LIN {X -176.622,Y -112.343,Z 160.000,A 0.000,B 0.000,C 180.000,E1 0.000} C_DIS
LIN {X -182.169,Y -103.103,Z 160.000,A 0.000,B 0.000,C 180.000,E1 0.000} C_DIS
LIN {X -187.236,Y -93.587,Z 160.000,A 0.000,B 0.000,C 180.000,E1 0.000} C_DIS
LIN {X -191.804,Y -83.827,Z 160.000,A 0.000,B 0.000,C 180.000,E1 0.000} C_DIS
LIN {X -195.867,Y -73.837,Z 160.000,A 0.000,B 0.000,C 180.000,E1 0.000} C_DIS
LIN {X -199.408,Y -63.658,Z 160.000,A 0.000,B 0.000,C 180.000,E1 0.000} C_DIS
LIN {X -202.421,Y -53.309,Z 160.000,A 0.000,B 0.000,C 180.000,E1 0.000} C_DIS
LIN {X -204.896,Y -42.818,Z 160.000,A 0.000,B 0.000,C 180.000,E1 0.000} C_DIS
LIN {X -206.829,Y -32.213,Z 160.000,A 0.000,B 0.000,C 180.000,E1 0.000} C_DIS
LIN {X -208.213,Y -21.523,Z 160.000,A 0.000,B 0.000,C 180.000,E1 0.000} C_DIS
LIN {X -208.336,Y -19.932,Z 160.000,A 0.000,B 0.000,C 180.000,E1 0.000} C_DIS
LIN {X 19.906,Y 208.310,Z 160.000,A 0.000,B 0.000,C 180.000,E1 0.000} C_DIS
;rapid-leaky
$VEL.CP=0.3
LIN {X -233.236,Y -36.326,Z 170.000,A 0.000,B 0.000,C 180.000,E1 0.000} C_DIS
;bead-perimeter_outer
$VEL.CP=0.59
LIN {X -231.057,Y -48.285,Z 170.000,A 0.000,B 0.000,C 180.000,E1 0.000} C_DIS
LIN {X -228.265,Y -60.113,Z 170.000,A 0.000,B 0.000,C 180.000,E1 0.000} C_DIS
LIN {X -224.866,Y -71.785,Z 170.000,A 0.000,B 0.000,C 180.000,E1 0.000} C_DIS
LIN {X -220.874,Y -83.267,Z 170.000,A 0.000,B 0.000,C 180.000,E1 0.000} C_DIS
LIN {X -216.295,Y -94.525,Z 170.000,A 0.000,B 0.000,C 180.000,E1 0.000} C_DIS
LIN {X -211.142,Y -105.535,Z 170.000,A 0.000,B 0.000,C 180.000,E1 0.000} C_DIS
LIN {X -205.429,Y -116.265,Z 170.000,A 0.000,B 0.000,C 180.000,E1 0.000} C_DIS
LIN {X -199.171,Y -126.685,Z 170.000,A 0.000,B 0.000,C 180.000,E1 0.000} C_DIS
LIN {X -192.385,Y -136.770,Z 170.000,A 0.000,B 0.000,C 180.000,E1 0.000} C_DIS
LIN {X -185.089,Y -146.493,Z 170.000,A 0.000,B 0.000,C 180.000,E1 0.000} C_DIS
LIN {X -177.303,Y -155.828,Z 170.000,A 0.000,B 0.000,C 180.000,E1 0.000} C_DIS
LIN {X -169.045,Y -164.748,Z 170.000,A 0.000,B 0.000,C 180.000,E1 0.000} C_DIS
LIN {X -160.340,Y -173.232,Z 170.000,A 0.000,B 0.000,C 180.000,E1 0.000} C_DIS
LIN {X -151.211,Y -181.256,Z 170.000,A 0.000,B 0.000,C 180.000,E1 0.000} C_DIS
LIN {X -141.679,Y -188.800,Z 170.000,A 0.000,B 0.000,C 180.000,E1 0.000} C_DIS
LIN {X -131.772,Y -195.844,Z 170.000,A 0.000,B 0.000,C 180.000,E1 0.000} C_DIS
LIN {X -121.516,Y -202.367,Z 170.000,A 0.000,B 0.000,C 180.000,E1 0.000} C_DIS
LIN {X -110.937,Y -208.354,Z 170.000,A 0.000,B 0.000,C 180.000,E1 0.000} C_DIS
LIN {X -100.064,Y -213.788,Z 170.000,A 0.000,B 0.000,C 180.000,E1 0.000} C_DIS
LIN {X -88.925,Y -218.657,Z 170.000,A 0.000,B 0.000,C 180.000,E1 0.000} C_DIS
LIN {X -77.552,Y -222.945,Z 170.000,A 0.000,B 0.000,C 180.000,E1 0.000} C_DIS
LIN {X -65.972,Y -226.641,Z 170.000,A 0.000,B 0.000,C 180.000,E1 0.000} C_DIS
LIN {X -54.217,Y -229.736,Z 170.000,A 0.000,B 0.000,C 180.000,E1 0.000} C_DIS
LIN {X -42.318,Y -232.223,Z 170.000,A 0.000,B 0.000,C 180.000,E1 0.000} C_DIS
LIN {X -30.307,Y -234.093,Z 170.000,A 0.000,B 0.000,C 180.000,E1 0.000} C_DIS
LIN {X -18.217,Y -235.343,Z 170.000,A 0.000,B 0.000,C 180.000,E1 0.000} C_DIS
LIN {X -6.078,Y -235.969,Z 170.000,A 0.000,B 0.000,C 180.000,E1 0.000} C_DIS
LIN {X 6.078,Y -235.969,Z 170.000,A 0.000,B 0.000,C 180.000,E1 0.000} C_DIS
LIN {X 17.057,Y -235.404,Z 170.000,A 0.000,B 0.000,C 180.000,E1 0.000} C_DIS
LIN {X 18.215,Y -235.344,Z 170.000,A 0.000,B 0.000,C 180.000,E1 0.000} C_DIS
LIN {X 30.307,Y -234.093,Z 170.000,A 0.000,B 0.000,C 180.000,E1 0.000} C_DIS
LIN {X 42.318,Y -232.223,Z 170.000,A 0.000,B 0.000,C 180.000,E1 0.000} C_DIS
LIN {X 54.217,Y -229.736,Z 170.000,A 0.000,B 0.000,C 180.000,E1 0.000} C_DIS
LIN {X 65.972,Y -226.641,Z 170.000,A 0.000,B 0.000,C 180.000,E1 0.000} C_DIS
LIN {X 77.552,Y -222.945,Z 170.000,A 0.000,B 0.000,C 180.000,E1 0.000} C_DIS
LIN {X 88.925,Y -218.657,Z 170.000,A 0.000,B 0.000,C 180.000,E1 0.000} C_DIS
LIN {X 100.064,Y -213.788,Z 170.000,A 0.000,B 0.000,C 180.000,E1 0.000} C_DIS
LIN {X 110.937,Y -208.354,Z 170.000,A 0.000,B 0.000,C 180.000,E1 0.000} C_DIS
LIN {X 121.516,Y -202.367,Z 170.000,A 0.000,B 0.000,C 180.000,E1 0.000} C_DIS
LIN {X 131.772,Y -195.844,Z 170.000,A 0.000,B 0.000,C 180.000,E1 0.000} C_DIS
LIN {X 141.679,Y -188.800,Z 170.000,A 0.000,B 0.000,C 180.000,E1 0.000} C_DIS
LIN {X 151.211,Y -181.256,Z 170.000,A 0.000,B 0.000,C 180.000,E1 0.000} C_DIS
LIN {X 160.340,Y -173.232,Z 170.000,A 0.000,B 0.000,C 180.000,E1 0.000} C_DIS
LIN {X 169.045,Y -164.748,Z 170.000,A 0.000,B 0.000,C 180.000,E1 0.000} C_DIS
LIN {X 177.303,Y -155.828,Z 170.000,A 0.000,B 0.000,C 180.000,E1 0.000} C_DIS
LIN {X 185.089,Y -146.493,Z 170.000,A 0.000,B 0.000,C 180.000,E1 0.000} C_DIS
LIN {X 192.385,Y -136.770,Z 170.000,A 0.000,B 0.000,C 180.000,E1 0.000} C_DIS
LIN {X 199.171,Y -126.685,Z 170.000,A 0.000,B 0.000,C 180.000,E1 0.000} C_DIS
LIN {X 205.429,Y -116.265,Z 170.000,A 0.000,B 0.000,C 180.000,E1 0.000} C_DIS
LIN {X 211.142,Y -105.535,Z 170.000,A 0.000,B 0.000,C 180.000,E1 0.000} C_DIS
LIN {X 216.295,Y -94.525,Z 170.000,A 0.000,B 0.000,C 180.000,E1 0.000} C_DIS
LIN {X 220.874,Y -83.267,Z 170.000,A 0.000,B 0.000,C 180.000,E1 0.000} C_DIS
LIN {X 224.866,Y -71.785,Z 170.000,A 0.000,B 0.000,C 180.000,E1 0.000} C_DIS
LIN {X 228.265,Y -60.113,Z 170.000,A 0.000,B 0.000,C 180.000,E1 0.000} C_DIS
LIN {X 231.057,Y -48.285,Z 170.000,A 0.000,B 0.000,C 180.000,E1 0.000} C_DIS
LIN {X 233.236,Y -36.326,Z 170.000,A 0.000,B 0.000,C 180.000,E1 0.000} C_DIS
LIN {X 234.796,Y -24.271,Z 170.000,A 0.000,B 0.000,C 180.000,E1 0.000} C_DIS
LIN {X 235.735,Y -12.151,Z 170.000,A 0.000,B 0.000,C 180.000,E1 0.000} C_DIS
LIN {X 236.047,Y 0.000,Z 170.000,A 0.000,B 0.000,C 180.000,E1 0.000} C_DIS
LIN {X 235.735,Y 12.151,Z 170.000,A 0.000,B 0.000,C 180.000,E1 0.000} C_DIS
LIN {X 234.796,Y 24.271,Z 170.000,A 0.000,B 0.000,C 180.000,E1 0.000} C_DIS
LIN {X 233.236,Y 36.326,Z 170.000,A 0.000,B 0.000,C 180.000,E1 0.000} C_DIS
LIN {X 231.057,Y 48.285,Z 170.000,A 0.000,B 0.000,C 180.000,E1 0.000} C_DIS
LIN {X 228.265,Y 60.113,Z 170.000,A 0.000,B 0.000,C 180.000,E1 0.000} C_DIS
LIN {X 224.866,Y 71.785,Z 170.000,A 0.000,B 0.000,C 180.000,E1 0.000} C_DIS
LIN {X 220.874,Y 83.267,Z 170.000,A 0.000,B 0.000,C 180.000,E1 0.000} C_DIS
LIN {X 216.295,Y 94.525,Z 170.000,A 0.000,B 0.000,C 180.000,E1 0.000} C_DIS
LIN {X 211.142,Y 105.535,Z 170.000,A 0.000,B 0.000,C 180.000,E1 0.000} C_DIS
LIN {X 205.429,Y 116.265,Z 170.000,A 0.000,B 0.000,C 180.000,E1 0.000} C_DIS
LIN {X 199.171,Y 126.685,Z 170.000,A 0.000,B 0.000,C 180.000,E1 0.000} C_DIS
LIN {X 192.385,Y 136.770,Z 170.000,A 0.000,B 0.000,C 180.000,E1 0.000} C_DIS
LIN {X 185.089,Y 146.493,Z 170.000,A 0.000,B 0.000,C 180.000,E1 0.000} C_DIS
LIN {X 177.303,Y 155.828,Z 170.000,A 0.000,B 0.000,C 180.000,E1 0.000} C_DIS
LIN {X 169.045,Y 164.748,Z 170.000,A 0.000,B 0.000,C 180.000,E1 0.000} C_DIS
LIN {X 160.340,Y 173.232,Z 170.000,A 0.000,B 0.000,C 180.000,E1 0.000} C_DIS
LIN {X 151.211,Y 181.256,Z 170.000,A 0.000,B 0.000,C 180.000,E1 0.000} C_DIS
LIN {X 141.679,Y 188.800,Z 170.000,A 0.000,B 0.000,C 180.000,E1 0.000} C_DIS
LIN {X 131.772,Y 195.844,Z 170.000,A 0.000,B 0.000,C 180.000,E1 0.000} C_DIS
LIN {X 121.516,Y 202.367,Z 170.000,A 0.000,B 0.000,C 180.000,E1 0.000} C_DIS
LIN {X 110.937,Y 208.354,Z 170.000,A 0.000,B 0.000,C 180.000,E1 0.000} C_DIS
LIN {X 100.064,Y 213.788,Z 170.000,A 0.000,B 0.000,C 180.000,E1 0.000} C_DIS
LIN {X 88.925,Y 218.657,Z 170.000,A 0.000,B 0.000,C 180.000,E1 0.000} C_DIS
LIN {X 77.552,Y 222.945,Z 170.000,A 0.000,B 0.000,C 180.000,E1 0.000} C_DIS
LIN {X 65.972,Y 226.641,Z 170.000,A 0.000,B 0.000,C 180.000,E1 0.000} C_DIS
LIN {X 54.217,Y 229.736,Z 170.000,A 0.000,B 0.000,C 180.000,E1 0.000} C_DIS
LIN {X 42.318,Y 232.223,Z 170.000,A 0.000,B 0.000,C 180.000,E1 0.000} C_DIS
LIN {X 30.307,Y 234.093,Z 170.000,A 0.000,B 0.000,C 180.000,E1 0.000} C_DIS
LIN {X 18.217,Y 235.343,Z 170.000,A 0.000,B 0.000,C 180.000,E1 0.000} C_DIS
LIN {X 6.078,Y 235.969,Z 170.000,A 0.000,B 0.000,C 180.000,E1 0.000} C_DIS
LIN {X -6.078,Y 235.969,Z 170.000,A 0.000,B 0.000,C 180.000,E1 0.000} C_DIS
LIN {X -18.215,Y 235.344,Z 170.000,A 0.000,B 0.000,C 180.000,E1 0.000} C_DIS
LIN {X -30.307,Y 234.093,Z 170.000,A 0.000,B 0.000,C 180.000,E1 0.000} C_DIS
LIN {X -42.318,Y 232.223,Z 170.000,A 0.000,B 0.000,C 180.000,E1 0.000} C_DIS
LIN {X -54.217,Y 229.736,Z 170.000,A 0.000,B 0.000,C 180.000,E1 0.000} C_DIS
LIN {X -65.972,Y 226.641,Z 170.000,A 0.000,B 0.000,C 180.000,E1 0.000} C_DIS
LIN {X -77.552,Y 222.945,Z 170.000,A 0.000,B 0.000,C 180.000,E1 0.000} C_DIS
LIN {X -88.925,Y 218.657,Z 170.000,A 0.000,B 0.000,C 180.000,E1 0.000} C_DIS
LIN {X -100.064,Y 213.788,Z 170.000,A 0.000,B 0.000,C 180.000,E1 0.000} C_DIS
LIN {X -110.937,Y 208.354,Z 170.000,A 0.000,B 0.000,C 180.000,E1 0.000} C_DIS
LIN {X -121.516,Y 202.367,Z 170.000,A 0.000,B 0.000,C 180.000,E1 0.000} C_DIS
LIN {X -131.772,Y 195.844,Z 170.000,A 0.000,B 0.000,C 180.000,E1 0.000} C_DIS
LIN {X -141.679,Y 188.800,Z 170.000,A 0.000,B 0.000,C 180.000,E1 0.000} C_DIS
LIN {X -151.211,Y 181.256,Z 170.000,A 0.000,B 0.000,C 180.000,E1 0.000} C_DIS
LIN {X -160.340,Y 173.232,Z 170.000,A 0.000,B 0.000,C 180.000,E1 0.000} C_DIS
LIN {X -169.045,Y 164.748,Z 170.000,A 0.000,B 0.000,C 180.000,E1 0.000} C_DIS
LIN {X -177.303,Y 155.828,Z 170.000,A 0.000,B 0.000,C 180.000,E1 0.000} C_DIS
LIN {X -185.089,Y 146.493,Z 170.000,A 0.000,B 0.000,C 180.000,E1 0.000} C_DIS
LIN {X -192.385,Y 136.770,Z 170.000,A 0.000,B 0.000,C 180.000,E1 0.000} C_DIS
LIN {X -199.171,Y 126.685,Z 170.000,A 0.000,B 0.000,C 180.000,E1 0.000} C_DIS
LIN {X -205.429,Y 116.265,Z 170.000,A 0.000,B 0.000,C 180.000,E1 0.000} C_DIS
LIN {X -211.142,Y 105.535,Z 170.000,A 0.000,B 0.000,C 180.000,E1 0.000} C_DIS
LIN {X -216.295,Y 94.525,Z 170.000,A 0.000,B 0.000,C 180.000,E1 0.000} C_DIS
LIN {X -220.874,Y 83.267,Z 170.000,A 0.000,B 0.000,C 180.000,E1 0.000} C_DIS
LIN {X -224.866,Y 71.785,Z 170.000,A 0.000,B 0.000,C 180.000,E1 0.000} C_DIS
LIN {X -228.265,Y 60.113,Z 170.000,A 0.000,B 0.000,C 180.000,E1 0.000} C_DIS
LIN {X -231.057,Y 48.285,Z 170.000,A 0.000,B 0.000,C 180.000,E1 0.000} C_DIS
LIN {X -233.236,Y 36.326,Z 170.000,A 0.000,B 0.000,C 180.000,E1 0.000} C_DIS
LIN {X -234.796,Y 24.271,Z 170.000,A 0.000,B 0.000,C 180.000,E1 0.000} C_DIS
LIN {X -235.735,Y 12.151,Z 170.000,A 0.000,B 0.000,C 180.000,E1 0.000} C_DIS
LIN {X -236.047,Y 0.000,Z 170.000,A 0.000,B 0.000,C 180.000,E1 0.000} C_DIS
LIN {X -235.735,Y -12.151,Z 170.000,A 0.000,B 0.000,C 180.000,E1 0.000} C_DIS
LIN {X -234.796,Y -24.271,Z 170.000,A 0.000,B 0.000,C 180.000,E1 0.000} C_DIS
LIN {X -233.236,Y -36.326,Z 170.000,A 0.000,B 0.000,C 180.000,E1 0.000} C_DIS
;rapid-leaky
$VEL.CP=0.3
LIN {X -217.875,Y -33.934,Z 170.000,A 0.000,B 0.000,C 180.000,E1 0.000} C_DIS
;bead-perimeter_inner
$VEL.CP=0.59
LIN {X -215.841,Y -45.105,Z 170.000,A 0.000,B 0.000,C 180.000,E1 0.000} C_DIS
LIN {X -213.232,Y -56.153,Z 170.000,A 0.000,B 0.000,C 180.000,E1 0.000} C_DIS
LIN {X -210.057,Y -67.058,Z 170.000,A 0.000,B 0.000,C 180.000,E1 0.000} C_DIS
LIN {X -206.328,Y -77.784,Z 170.000,A 0.000,B 0.000,C 180.000,E1 0.000} C_DIS
LIN {X -202.050,Y -88.300,Z 170.000,A 0.000,B 0.000,C 180.000,E1 0.000} C_DIS
LIN {X -197.237,Y -98.585,Z 170.000,A 0.000,B 0.000,C 180.000,E1 0.000} C_DIS
LIN {X -191.900,Y -108.608,Z 170.000,A 0.000,B 0.000,C 180.000,E1 0.000} C_DIS
LIN {X -186.055,Y -118.342,Z 170.000,A 0.000,B 0.000,C 180.000,E1 0.000} C_DIS
LIN {X -179.716,Y -127.763,Z 170.000,A 0.000,B 0.000,C 180.000,E1 0.000} C_DIS
LIN {X -172.900,Y -136.846,Z 170.000,A 0.000,B 0.000,C 180.000,E1 0.000} C_DIS
LIN {X -165.626,Y -145.566,Z 170.000,A 0.000,B 0.000,C 180.000,E1 0.000} C_DIS
LIN {X -157.913,Y -153.898,Z 170.000,A 0.000,B 0.000,C 180.000,E1 0.000} C_DIS
LIN {X -149.781,Y -161.824,Z 170.000,A 0.000,B 0.000,C 180.000,E1 0.000} C_DIS
LIN {X -141.253,Y -169.319,Z 170.000,A 0.000,B 0.000,C 180.000,E1 0.000} C_DIS
LIN {X -132.349,Y -176.367,Z 170.000,A 0.000,B 0.000,C 180.000,E1 0.000} C_DIS
LIN {X -123.095,Y -182.946,Z 170.000,A 0.000,B 0.000,C 180.000,E1 0.000} C_DIS
LIN {X -113.514,Y -189.039,Z 170.000,A 0.000,B 0.000,C 180.000,E1 0.000} C_DIS
LIN {X -103.631,Y -194.633,Z 170.000,A 0.000,B 0.000,C 180.000,E1 0.000} C_DIS
LIN {X -93.474,Y -199.709,Z 170.000,A 0.000,B 0.000,C 180.000,E1 0.000} C_DIS
LIN {X -83.068,Y -204.257,Z 170.000,A 0.000,B 0.000,C 180.000,E1 0.000} C_DIS
LIN {X -72.445,Y -208.262,Z 170.000,A 0.000,B 0.000,C 180.000,E1 0.000} C_DIS
LIN {X -61.628,Y -211.715,Z 170.000,A 0.000,B 0.000,C 180.000,E1 0.000} C_DIS
LIN {X -50.647,Y -214.607,Z 170.000,A 0.000,B 0.000,C 180.000,E1 0.000} C_DIS
LIN {X -39.532,Y -216.930,Z 170.000,A 0.000,B 0.000,C 180.000,E1 0.000} C_DIS
LIN {X -28.312,Y -218.677,Z 170.000,A 0.000,B 0.000,C 180.000,E1 0.000} C_DIS
LIN {X -17.017,Y -219.845,Z 170.000,A 0.000,B 0.000,C 180.000,E1 0.000} C_DIS
LIN {X -5.678,Y -220.429,Z 170.000,A 0.000,B 0.000,C 180.000,E1 0.000} C_DIS
LIN {X 5.679,Y -220.429,Z 170.000,A 0.000,B 0.000,C 180.000,E1 0.000} C_DIS
LIN {X 16.253,Y -219.885,Z 170.000,A 0.000,B 0.000,C 180.000,E1 0.000} C_DIS
LIN {X 17.011,Y -219.845,Z 170.000,A 0.000,B 0.000,C 180.000,E1 0.000} C_DIS
LIN {X 28.312,Y -218.677,Z 170.000,A 0.000,B 0.000,C 180.000,E1 0.000} C_DIS
LIN {X 39.532,Y -216.930,Z 170.000,A 0.000,B 0.000,C 180.000,E1 0.000} C_DIS
LIN {X 50.647,Y -214.607,Z 170.000,A 0.000,B 0.000,C 180.000,E1 0.000} C_DIS
LIN {X 61.628,Y -211.715,Z 170.000,A 0.000,B 0.000,C 180.000,E1 0.000} C_DIS
LIN {X 72.445,Y -208.262,Z 170.000,A 0.000,B 0.000,C 180.000,E1 0.000} C_DIS
LIN {X 83.068,Y -204.257,Z 170.000,A 0.000,B 0.000,C 180.000,E1 0.000} C_DIS
LIN {X 93.474,Y -199.709,Z 170.000,A 0.000,B 0.000,C 180.000,E1 0.000} C_DIS
LIN {X 103.631,Y -194.633,Z 170.000,A 0.000,B 0.000,C 180.000,E1 0.000} C_DIS
LIN {X 113.514,Y -189.039,Z 170.000,A 0.000,B 0.000,C 180.000,E1 0.000} C_DIS
LIN {X 123.095,Y -182.946,Z 170.000,A 0.000,B 0.000,C 180.000,E1 0.000} C_DIS
LIN {X 132.349,Y -176.367,Z 170.000,A 0.000,B 0.000,C 180.000,E1 0.000} C_DIS
LIN {X 141.253,Y -169.319,Z 170.000,A 0.000,B 0.000,C 180.000,E1 0.000} C_DIS
LIN {X 149.781,Y -161.824,Z 170.000,A 0.000,B 0.000,C 180.000,E1 0.000} C_DIS
LIN {X 157.913,Y -153.898,Z 170.000,A 0.000,B 0.000,C 180.000,E1 0.000} C_DIS
LIN {X 165.626,Y -145.566,Z 170.000,A 0.000,B 0.000,C 180.000,E1 0.000} C_DIS
LIN {X 172.900,Y -136.846,Z 170.000,A 0.000,B 0.000,C 180.000,E1 0.000} C_DIS
LIN {X 179.716,Y -127.763,Z 170.000,A 0.000,B 0.000,C 180.000,E1 0.000} C_DIS
LIN {X 186.055,Y -118.342,Z 170.000,A 0.000,B 0.000,C 180.000,E1 0.000} C_DIS
LIN {X 191.900,Y -108.608,Z 170.000,A 0.000,B 0.000,C 180.000,E1 0.000} C_DIS
LIN {X 197.237,Y -98.585,Z 170.000,A 0.000,B 0.000,C 180.000,E1 0.000} C_DIS
LIN {X 202.050,Y -88.300,Z 170.000,A 0.000,B 0.000,C 180.000,E1 0.000} C_DIS
LIN {X 206.328,Y -77.784,Z 170.000,A 0.000,B 0.000,C 180.000,E1 0.000} C_DIS
LIN {X 210.057,Y -67.058,Z 170.000,A 0.000,B 0.000,C 180.000,E1 0.000} C_DIS
LIN {X 213.232,Y -56.153,Z 170.000,A 0.000,B 0.000,C 180.000,E1 0.000} C_DIS
LIN {X 215.841,Y -45.105,Z 170.000,A 0.000,B 0.000,C 180.000,E1 0.000} C_DIS
LIN {X 217.875,Y -33.934,Z 170.000,A 0.000,B 0.000,C 180.000,E1 0.000} C_DIS
LIN {X 219.334,Y -22.672,Z 170.000,A 0.000,B 0.000,C 180.000,E1 0.000} C_DIS
LIN {X 220.210,Y -11.351,Z 170.000,A 0.000,B 0.000,C 180.000,E1 0.000} C_DIS
LIN {X 220.502,Y 0.000,Z 170.000,A 0.000,B 0.000,C 180.000,E1 0.000} C_DIS
LIN {X 220.210,Y 11.351,Z 170.000,A 0.000,B 0.000,C 180.000,E1 0.000} C_DIS
LIN {X 219.334,Y 22.672,Z 170.000,A 0.000,B 0.000,C 180.000,E1 0.000} C_DIS
LIN {X 217.875,Y 33.934,Z 170.000,A 0.000,B 0.000,C 180.000,E1 0.000} C_DIS
LIN {X 215.841,Y 45.105,Z 170.000,A 0.000,B 0.000,C 180.000,E1 0.000} C_DIS
LIN {X 213.232,Y 56.153,Z 170.000,A 0.000,B 0.000,C 180.000,E1 0.000} C_DIS
LIN {X 210.057,Y 67.058,Z 170.000,A 0.000,B 0.000,C 180.000,E1 0.000} C_DIS
LIN {X 206.328,Y 77.784,Z 170.000,A 0.000,B 0.000,C 180.000,E1 0.000} C_DIS
LIN {X 202.050,Y 88.300,Z 170.000,A 0.000,B 0.000,C 180.000,E1 0.000} C_DIS
LIN {X 197.237,Y 98.585,Z 170.000,A 0.000,B 0.000,C 180.000,E1 0.000} C_DIS
LIN {X 191.900,Y 108.608,Z 170.000,A 0.000,B 0.000,C 180.000,E1 0.000} C_DIS
LIN {X 186.055,Y 118.342,Z 170.000,A 0.000,B 0.000,C 180.000,E1 0.000} C_DIS
LIN {X 179.716,Y 127.763,Z 170.000,A 0.000,B 0.000,C 180.000,E1 0.000} C_DIS
LIN {X 172.900,Y 136.846,Z 170.000,A 0.000,B 0.000,C 180.000,E1 0.000} C_DIS
LIN {X 165.626,Y 145.566,Z 170.000,A 0.000,B 0.000,C 180.000,E1 0.000} C_DIS
LIN {X 157.913,Y 153.898,Z 170.000,A 0.000,B 0.000,C 180.000,E1 0.000} C_DIS
LIN {X 149.781,Y 161.824,Z 170.000,A 0.000,B 0.000,C 180.000,E1 0.000} C_DIS
LIN {X 141.253,Y 169.319,Z 170.000,A 0.000,B 0.000,C 180.000,E1 0.000} C_DIS
LIN {X 132.349,Y 176.367,Z 170.000,A 0.000,B 0.000,C 180.000,E1 0.000} C_DIS
LIN {X 123.095,Y 182.946,Z 170.000,A 0.000,B 0.000,C 180.000,E1 0.000} C_DIS
LIN {X 113.514,Y 189.039,Z 170.000,A 0.000,B 0.000,C 180.000,E1 0.000} C_DIS
LIN {X 103.631,Y 194.633,Z 170.000,A 0.000,B 0.000,C 180.000,E1 0.000} C_DIS
LIN {X 93.474,Y 199.709,Z 170.000,A 0.000,B 0.000,C 180.000,E1 0.000} C_DIS
LIN {X 83.068,Y 204.257,Z 170.000,A 0.000,B 0.000,C 180.000,E1 0.000} C_DIS
LIN {X 72.445,Y 208.262,Z 170.000,A 0.000,B 0.000,C 180.000,E1 0.000} C_DIS
LIN {X 61.628,Y 211.715,Z 170.000,A 0.000,B 0.000,C 180.000,E1 0.000} C_DIS
LIN {X 50.647,Y 214.607,Z 170.000,A 0.000,B 0.000,C 180.000,E1 0.000} C_DIS
LIN {X 39.532,Y 216.930,Z 170.000,A 0.000,B 0.000,C 180.000,E1 0.000} C_DIS
LIN {X 28.312,Y 218.677,Z 170.000,A 0.000,B 0.000,C 180.000,E1 0.000} C_DIS
LIN {X 17.017,Y 219.845,Z 170.000,A 0.000,B 0.000,C 180.000,E1 0.000} C_DIS
LIN {X 5.678,Y 220.429,Z 170.000,A 0.000,B 0.000,C 180.000,E1 0.000} C_DIS
LIN {X -5.679,Y 220.429,Z 170.000,A 0.000,B 0.000,C 180.000,E1 0.000} C_DIS
LIN {X -17.011,Y 219.845,Z 170.000,A 0.000,B 0.000,C 180.000,E1 0.000} C_DIS
LIN {X -28.312,Y 218.677,Z 170.000,A 0.000,B 0.000,C 180.000,E1 0.000} C_DIS
LIN {X -39.532,Y 216.930,Z 170.000,A 0.000,B 0.000,C 180.000,E1 0.000} C_DIS
LIN {X -50.647,Y 214.607,Z 170.000,A 0.000,B 0.000,C 180.000,E1 0.000} C_DIS
LIN {X -61.628,Y 211.715,Z 170.000,A 0.000,B 0.000,C 180.000,E1 0.000} C_DIS
LIN {X -72.445,Y 208.262,Z 170.000,A 0.000,B 0.000,C 180.000,E1 0.000} C_DIS
LIN {X -83.068,Y 204.257,Z 170.000,A 0.000,B 0.000,C 180.000,E1 0.000} C_DIS
LIN {X -93.474,Y 199.709,Z 170.000,A 0.000,B 0.000,C 180.000,E1 0.000} C_DIS
LIN {X -103.631,Y 194.633,Z 170.000,A 0.000,B 0.000,C 180.000,E1 0.000} C_DIS
LIN {X -113.514,Y 189.039,Z 170.000,A 0.000,B 0.000,C 180.000,E1 0.000} C_DIS
LIN {X -123.095,Y 182.946,Z 170.000,A 0.000,B 0.000,C 180.000,E1 0.000} C_DIS
LIN {X -132.349,Y 176.367,Z 170.000,A 0.000,B 0.000,C 180.000,E1 0.000} C_DIS
LIN {X -141.253,Y 169.319,Z 170.000,A 0.000,B 0.000,C 180.000,E1 0.000} C_DIS
LIN {X -149.781,Y 161.824,Z 170.000,A 0.000,B 0.000,C 180.000,E1 0.000} C_DIS
LIN {X -157.913,Y 153.898,Z 170.000,A 0.000,B 0.000,C 180.000,E1 0.000} C_DIS
LIN {X -165.626,Y 145.566,Z 170.000,A 0.000,B 0.000,C 180.000,E1 0.000} C_DIS
LIN {X -172.900,Y 136.846,Z 170.000,A 0.000,B 0.000,C 180.000,E1 0.000} C_DIS
LIN {X -179.716,Y 127.763,Z 170.000,A 0.000,B 0.000,C 180.000,E1 0.000} C_DIS
LIN {X -186.055,Y 118.342,Z 170.000,A 0.000,B 0.000,C 180.000,E1 0.000} C_DIS
LIN {X -191.900,Y 108.608,Z 170.000,A 0.000,B 0.000,C 180.000,E1 0.000} C_DIS
LIN {X -197.237,Y 98.585,Z 170.000,A 0.000,B 0.000,C 180.000,E1 0.000} C_DIS
LIN {X -202.050,Y 88.300,Z 170.000,A 0.000,B 0.000,C 180.000,E1 0.000} C_DIS
LIN {X -206.328,Y 77.784,Z 170.000,A 0.000,B 0.000,C 180.000,E1 0.000} C_DIS
LIN {X -210.057,Y 67.058,Z 170.000,A 0.000,B 0.000,C 180.000,E1 0.000} C_DIS
LIN {X -213.232,Y 56.153,Z 170.000,A 0.000,B 0.000,C 180.000,E1 0.000} C_DIS
LIN {X -215.841,Y 45.105,Z 170.000,A 0.000,B 0.000,C 180.000,E1 0.000} C_DIS
LIN {X -217.875,Y 33.934,Z 170.000,A 0.000,B 0.000,C 180.000,E1 0.000} C_DIS
LIN {X -219.334,Y 22.672,Z 170.000,A 0.000,B 0.000,C 180.000,E1 0.000} C_DIS
LIN {X -220.210,Y 11.351,Z 170.000,A 0.000,B 0.000,C 180.000,E1 0.000} C_DIS
LIN {X -220.502,Y 0.000,Z 170.000,A 0.000,B 0.000,C 180.000,E1 0.000} C_DIS
LIN {X -220.210,Y -11.351,Z 170.000,A 0.000,B 0.000,C 180.000,E1 0.000} C_DIS
LIN {X -219.334,Y -22.672,Z 170.000,A 0.000,B 0.000,C 180.000,E1 0.000} C_DIS
LIN {X -217.875,Y -33.934,Z 170.000,A 0.000,B 0.000,C 180.000,E1 0.000} C_DIS
;rapid-leaky
$VEL.CP=0.3
LIN {X -202.207,Y 13.804,Z 170.000,A 0.000,B 0.000,C 180.000,E1 0.000} C_DIS
;bead-sparse_infill
$VEL.CP=0.59
LIN {X 13.823,Y -202.226,Z 170.000,A 0.000,B 0.000,C 180.000,E1 0.000} C_DIS
LIN {X 15.337,Y -202.148,Z 170.000,A 0.000,B 0.000,C 180.000,E1 0.000} C_DIS
LIN {X 15.636,Y -202.133,Z 170.000,A 0.000,B 0.000,C 180.000,E1 0.000} C_DIS
LIN {X 26.031,Y -201.058,Z 170.000,A 0.000,B 0.000,C 180.000,E1 0.000} C_DIS
LIN {X 36.347,Y -199.452,Z 170.000,A 0.000,B 0.000,C 180.000,E1 0.000} C_DIS
LIN {X 46.566,Y -197.316,Z 170.000,A 0.000,B 0.000,C 180.000,E1 0.000} C_DIS
LIN {X 56.663,Y -194.657,Z 170.000,A 0.000,B 0.000,C 180.000,E1 0.000} C_DIS
LIN {X 66.608,Y -191.483,Z 170.000,A 0.000,B 0.000,C 180.000,E1 0.000} C_DIS
LIN {X 76.375,Y -187.800,Z 170.000,A 0.000,B 0.000,C 180.000,E1 0.000} C_DIS
LIN {X 85.943,Y -183.618,Z 170.000,A 0.000,B 0.000,C 180.000,E1 0.000} C_DIS
LIN {X 95.281,Y -178.951,Z 170.000,A 0.000,B 0.000,C 180.000,E1 0.000} C_DIS
LIN {X 104.369,Y -173.808,Z 170.000,A 0.000,B 0.000,C 180.000,E1 0.000} C_DIS
LIN {X 113.177,Y -168.206,Z 170.000,A 0.000,B 0.000,C 180.000,E1 0.000} C_DIS
LIN {X 121.685,Y -162.157,Z 170.000,A 0.000,B 0.000,C 180.000,E1 0.000} C_DIS
LIN {X 126.735,Y -158.160,Z 170.000,A 0.000,B 0.000,C 180.000,E1 0.000} C_DIS
LIN {X -158.186,Y 126.760,Z 170.000,A 0.000,B 0.000,C 180.000,E1 0.000} C_DIS
LIN {X -152.282,Y 133.837,Z 170.000,A 0.000,B 0.000,C 180.000,E1 0.000} C_DIS
LIN {X -145.190,Y 141.499,Z 170.000,A 0.000,B 0.000,C 180.000,E1 0.000} C_DIS
LIN {X -137.713,Y 148.786,Z 170.000,A 0.000,B 0.000,C 180.000,E1 0.000} C_DIS
LIN {X -129.872,Y 155.677,Z 170.000,A 0.000,B 0.000,C 180.000,E1 0.000} C_DIS
LIN {X -121.685,Y 162.157,Z 170.000,A 0.000,B 0.000,C 180.000,E1 0.000} C_DIS
LIN {X -113.177,Y 168.206,Z 170.000,A 0.000,B 0.000,C 180.000,E1 0.000} C_DIS
LIN {X -104.369,Y 173.808,Z 170.000,A 0.000,B 0.000,C 180.000,E1 0.000} C_DIS
LIN {X -95.281,Y 178.951,Z 170.000,A 0.000,B 0.000,C 180.000,E1 0.000} C_DIS
LIN {X -85.943,Y 183.618,Z 170.000,A 0.000,B 0.000,C 180.000,E1 0.000} C_DIS
LIN {X -76.375,Y 187.800,Z 170.000,A 0.000,B 0.000,C 180.000,E1 0.000} C_DIS
LIN {X -66.608,Y 191.483,Z 170.000,A 0.000,B 0.000,C 180.000,E1 0.000} C_DIS
LIN {X -66.095,Y 191.646,Z 170.000,A 0.000,B 0.000,C 180.000,E1 0.000} C_DIS
LIN {X 191.604,Y -66.052,Z 170.000,A 0.000,B 0.000,C 180.000,E1 0.000} C_DIS
LIN {X 193.133,Y -61.656,Z 170.000,A 0.000,B 0.000,C 180.000,E1 0.000} C_DIS
LIN {X 196.053,Y -51.628,Z 170.000,A 0.000,B 0.000,C 180.000,E1 0.000} C_DIS
LIN {X 198.450,Y -41.471,Z 170.000,A 0.000,B 0.000,C 180.000,E1 0.000} C_DIS
LIN {X 200.321,Y -31.201,Z 170.000,A 0.000,B 0.000,C 180.000,E1 0.000} C_DIS
LIN {X 201.662,Y -20.845,Z 170.000,A 0.000,B 0.000,C 180.000,E1 0.000} C_DIS
LIN {X 202.468,Y -10.437,Z 170.000,A 0.000,B 0.000,C 180.000,E1 0.000} C_DIS
LIN {X 202.736,Y 0.000,Z 170.000,A 0.000,B 0.000,C 180.000,E1 0.000} C_DIS
LIN {X 202.468,Y 10.437,Z 170.000,A 0.000,B 0.000,C 180.000,E1 0.000} C_DIS
LIN {X 201.662,Y 20.845,Z 170.000,A 0.000,B 0.000,C 180.000,E1 0.000} C_DIS
LIN {X 200.321,Y 31.201,Z 170.000,A 0.000,B 0.000,C 180.000,E1 0.000} C_DIS
LIN {X 198.450,Y 41.471,Z 170.000,A 0.000,B 0.000,C 180.000,E1 0.000} C_DIS
LIN {X 196.053,Y 51.628,Z 170.000,A 0.000,B 0.000,C 180.000,E1 0.000} C_DIS
LIN {X 193.133,Y 61.656,Z 170.000,A 0.000,B 0.000,C 180.000,E1 0.000} C_DIS
LIN {X 189.704,Y 71.517,Z 170.000,A 0.000,B 0.000,C 180.000,E1 0.000} C_DIS
LIN {X 185.771,Y 81.185,Z 170.000,A 0.000,B 0.000,C 180.000,E1 0.000} C_DIS
LIN {X 181.345,Y 90.642,Z 170.000,A 0.000,B 0.000,C 180.000,E1 0.000} C_DIS
LIN {X 176.439,Y 99.857,Z 170.000,A 0.000,B 0.000,C 180.000,E1 0.000} C_DIS
LIN {X 171.064,Y 108.807,Z 170.000,A 0.000,B 0.000,C 180.000,E1 0.000} C_DIS
LIN {X 165.597,Y 116.933,Z 170.000,A 0.000,B 0.000,C 180.000,E1 0.000} C_DIS
LIN {X 117.144,Y 165.385,Z 170.000,A 0.000,B 0.000,C 180.000,E1 0.000} C_DIS
;rapid-leaky
$VEL.CP=0.3
LIN {X 5.890,Y -228.708,Z 180.000,A 0.000,B 0.000,C 180.000,E1 0.000} C_DIS
;bead-perimeter_outer
$VEL.CP=0.54
LIN {X 17.657,Y -228.101,Z 180.000,A 0.000,B 0.000,C 180.000,E1 0.000} C_DIS
LIN {X 29.375,Y -226.890,Z 180.000,A 0.000,B 0.000,C 180.000,E1 0.000} C_DIS
LIN {X 41.016,Y -225.077,Z 180.000,A 0.000,B 0.000,C 180.000,E1 0.000} C_DIS
LIN {X 52.549,Y -222.667,Z 180.000,A 0.000,B 0.000,C 180.000,E1 0.000} C_DIS
LIN {X 63.942,Y -219.667,Z 180.000,A 0.000,B 0.000,C 180.000,E1 0.000} C_DIS
LIN {X 75.165,Y -216.084,Z 180.000,A 0.000,B 0.000,C 180.000,E1 0.000} C_DIS
LIN {X 86.189,Y -211.927,Z 180.000,A 0.000,B 0.000,C 180.000,E1 0.000} C_DIS
LIN {X 96.983,Y -207.210,Z 180.000,A 0.000,B 0.000,C 180.000,E1 0.000} C_DIS
LIN {X 107.524,Y -201.942,Z 180.000,A 0.000,B 0.000,C 180.000,E1 0.000} C_DIS
LIN {X 117.777,Y -196.140,Z 180.000,A 0.000,B 0.000,C 180.000,E1 0.000} C_DIS
LIN {X 127.717,Y -189.817,Z 180.000,A 0.000,B 0.000,C 180.000,E1 0.000} C_DIS
LIN {X 137.318,Y -182.990,Z 180.000,A 0.000,B 0.000,C 180.000,E1 0.000} C_DIS
LIN {X 146.558,Y -175.677,Z 180.000,A 0.000,B 0.000,C 180.000,E1 0.000} C_DIS
LIN {X 155.407,Y -167.901,Z 180.000,A 0.000,B 0.000,C 180.000,E1 0.000} C_DIS
LIN {X 163.844,Y -159.678,Z 180.000,A 0.000,B 0.000,C 180.000,E1 0.000} C_DIS
LIN {X 171.846,Y -151.032,Z 180.000,A 0.000,B 0.000,C 180.000,E1 0.000} C_DIS
LIN {X 179.393,Y -141.985,Z 180.000,A 0.000,B 0.000,C 180.000,E1 0.000} C_DIS
LIN {X 186.465,Y -132.562,Z 180.000,A 0.000,B 0.000,C 180.000,E1 0.000} C_DIS
LIN {X 193.042,Y -122.788,Z 180.000,A 0.000,B 0.000,C 180.000,E1 0.000} C_DIS
LIN {X 199.107,Y -112.687,Z 180.000,A 0.000,B 0.000,C 180.000,E1 0.000} C_DIS
LIN {X 204.645,Y -102.287,Z 180.000,A 0.000,B 0.000,C 180.000,E1 0.000} C_DIS
LIN {X 209.638,Y -91.618,Z 180.000,A 0.000,B 0.000,C 180.000,E1 0.000} C_DIS
LIN {X 214.077,Y -80.704,Z 180.000,A 0.000,B 0.000,C 180.000,E1 0.000} C_DIS
LIN {X 217.947,Y -69.576,Z 180.000,A 0.000,B 0.000,C 180.000,E1 0.000} C_DIS
LIN {X 221.240,Y -58.264,Z 180.000,A 0.000,B 0.000,C 180.000,E1 0.000} C_DIS
LIN {X 223.946,Y -46.798,Z 180.000,A 0.000,B 0.000,C 180.000,E1 0.000} C_DIS
LIN {X 226.059,Y -35.207,Z 180.000,A 0.000,B 0.000,C 180.000,E1 0.000} C_DIS
LIN {X 227.571,Y -23.524,Z 180.000,A 0.000,B 0.000,C 180.000,E1 0.000} C_DIS
LIN {X 228.480,Y -11.777,Z 180.000,A 0.000,B 0.000,C 180.000,E1 0.000} C_DIS
LIN {X 228.784,Y 0.000,Z 180.000,A 0.000,B 0.000,C 180.000,E1 0.000} C_DIS
LIN {X 228.480,Y 11.777,Z 180.000,A 0.000,B 0.000,C 180.000,E1 0.000} C_DIS
LIN {X 227.571,Y 23.524,Z 180.000,A 0.000,B 0.000,C 180.000,E1 0.000} C_DIS
LIN {X 226.059,Y 35.207,Z 180.000,A 0.000,B 0.000,C 180.000,E1 0.000} C_DIS
LIN {X 223.946,Y 46.798,Z 180.000,A 0.000,B 0.000,C 180.000,E1 0.000} C_DIS
LIN {X 221.240,Y 58.264,Z 180.000,A 0.000,B 0.000,C 180.000,E1 0.000} C_DIS
LIN {X 217.947,Y 69.576,Z 180.000,A 0.000,B 0.000,C 180.000,E1 0.000} C_DIS
LIN {X 214.077,Y 80.704,Z 180.000,A 0.000,B 0.000,C 180.000,E1 0.000} C_DIS
LIN {X 209.638,Y 91.618,Z 180.000,A 0.000,B 0.000,C 180.000,E1 0.000} C_DIS
LIN {X 204.645,Y 102.287,Z 180.000,A 0.000,B 0.000,C 180.000,E1 0.000} C_DIS
LIN {X 199.107,Y 112.687,Z 180.000,A 0.000,B 0.000,C 180.000,E1 0.000} C_DIS
LIN {X 193.042,Y 122.788,Z 180.000,A 0.000,B 0.000,C 180.000,E1 0.000} C_DIS
LIN {X 186.465,Y 132.562,Z 180.000,A 0.000,B 0.000,C 180.000,E1 0.000} C_DIS
LIN {X 179.393,Y 141.985,Z 180.000,A 0.000,B 0.000,C 180.000,E1 0.000} C_DIS
LIN {X 171.846,Y 151.032,Z 180.000,A 0.000,B 0.000,C 180.000,E1 0.000} C_DIS
LIN {X 163.844,Y 159.678,Z 180.000,A 0.000,B 0.000,C 180.000,E1 0.000} C_DIS
LIN {X 155.407,Y 167.901,Z 180.000,A 0.000,B 0.000,C 180.000,E1 0.000} C_DIS
LIN {X 146.558,Y 175.677,Z 180.000,A 0.000,B 0.000,C 180.000,E1 0.000} C_DIS
LIN {X 137.318,Y 182.990,Z 180.000,A 0.000,B 0.000,C 180.000,E1 0.000} C_DIS
LIN {X 127.717,Y 189.817,Z 180.000,A 0.000,B 0.000,C 180.000,E1 0.000} C_DIS
LIN {X 117.777,Y 196.140,Z 180.000,A 0.000,B 0.000,C 180.000,E1 0.000} C_DIS
LIN {X 107.524,Y 201.942,Z 180.000,A 0.000,B 0.000,C 180.000,E1 0.000} C_DIS
LIN {X 96.984,Y 207.209,Z 180.000,A 0.000,B 0.000,C 180.000,E1 0.000} C_DIS
LIN {X 86.189,Y 211.928,Z 180.000,A 0.000,B 0.000,C 180.000,E1 0.000} C_DIS
LIN {X 75.165,Y 216.084,Z 180.000,A 0.000,B 0.000,C 180.000,E1 0.000} C_DIS
LIN {X 63.942,Y 219.667,Z 180.000,A 0.000,B 0.000,C 180.000,E1 0.000} C_DIS
LIN {X 52.549,Y 222.667,Z 180.000,A 0.000,B 0.000,C 180.000,E1 0.000} C_DIS
LIN {X 41.016,Y 225.077,Z 180.000,A 0.000,B 0.000,C 180.000,E1 0.000} C_DIS
LIN {X 29.375,Y 226.890,Z 180.000,A 0.000,B 0.000,C 180.000,E1 0.000} C_DIS
LIN {X 17.657,Y 228.101,Z 180.000,A 0.000,B 0.000,C 180.000,E1 0.000} C_DIS
LIN {X 5.890,Y 228.708,Z 180.000,A 0.000,B 0.000,C 180.000,E1 0.000} C_DIS
LIN {X -5.890,Y 228.708,Z 180.000,A 0.000,B 0.000,C 180.000,E1 0.000} C_DIS
LIN {X -17.657,Y 228.101,Z 180.000,A 0.000,B 0.000,C 180.000,E1 0.000} C_DIS
LIN {X -29.375,Y 226.890,Z 180.000,A 0.000,B 0.000,C 180.000,E1 0.000} C_DIS
LIN {X -41.016,Y 225.077,Z 180.000,A 0.000,B 0.000,C 180.000,E1 0.000} C_DIS
LIN {X -52.549,Y 222.667,Z 180.000,A 0.000,B 0.000,C 180.000,E1 0.000} C_DIS
LIN {X -63.942,Y 219.667,Z 180.000,A 0.000,B 0.000,C 180.000,E1 0.000} C_DIS
LIN {X -75.165,Y 216.084,Z 180.000,A 0.000,B 0.000,C 180.000,E1 0.000} C_DIS
LIN {X -86.189,Y 211.927,Z 180.000,A 0.000,B 0.000,C 180.000,E1 0.000} C_DIS
LIN {X -96.983,Y 207.210,Z 180.000,A 0.000,B 0.000,C 180.000,E1 0.000} C_DIS
LIN {X -107.524,Y 201.942,Z 180.000,A 0.000,B 0.000,C 180.000,E1 0.000} C_DIS
LIN {X -117.777,Y 196.140,Z 180.000,A 0.000,B 0.000,C 180.000,E1 0.000} C_DIS
LIN {X -127.717,Y 189.817,Z 180.000,A 0.000,B 0.000,C 180.000,E1 0.000} C_DIS
LIN {X -137.318,Y 182.990,Z 180.000,A 0.000,B 0.000,C 180.000,E1 0.000} C_DIS
LIN {X -146.558,Y 175.677,Z 180.000,A 0.000,B 0.000,C 180.000,E1 0.000} C_DIS
LIN {X -155.407,Y 167.901,Z 180.000,A 0.000,B 0.000,C 180.000,E1 0.000} C_DIS
LIN {X -163.844,Y 159.678,Z 180.000,A 0.000,B 0.000,C 180.000,E1 0.000} C_DIS
LIN {X -171.846,Y 151.032,Z 180.000,A 0.000,B 0.000,C 180.000,E1 0.000} C_DIS
LIN {X -179.393,Y 141.985,Z 180.000,A 0.000,B 0.000,C 180.000,E1 0.000} C_DIS
LIN {X -186.465,Y 132.562,Z 180.000,A 0.000,B 0.000,C 180.000,E1 0.000} C_DIS
LIN {X -193.042,Y 122.788,Z 180.000,A 0.000,B 0.000,C 180.000,E1 0.000} C_DIS
LIN {X -199.107,Y 112.687,Z 180.000,A 0.000,B 0.000,C 180.000,E1 0.000} C_DIS
LIN {X -204.645,Y 102.287,Z 180.000,A 0.000,B 0.000,C 180.000,E1 0.000} C_DIS
LIN {X -209.638,Y 91.618,Z 180.000,A 0.000,B 0.000,C 180.000,E1 0.000} C_DIS
LIN {X -214.077,Y 80.704,Z 180.000,A 0.000,B 0.000,C 180.000,E1 0.000} C_DIS
LIN {X -217.947,Y 69.576,Z 180.000,A 0.000,B 0.000,C 180.000,E1 0.000} C_DIS
LIN {X -221.240,Y 58.264,Z 180.000,A 0.000,B 0.000,C 180.000,E1 0.000} C_DIS
LIN {X -223.946,Y 46.798,Z 180.000,A 0.000,B 0.000,C 180.000,E1 0.000} C_DIS
LIN {X -226.059,Y 35.207,Z 180.000,A 0.000,B 0.000,C 180.000,E1 0.000} C_DIS
LIN {X -227.571,Y 23.524,Z 180.000,A 0.000,B 0.000,C 180.000,E1 0.000} C_DIS
LIN {X -228.480,Y 11.777,Z 180.000,A 0.000,B 0.000,C 180.000,E1 0.000} C_DIS
LIN {X -228.784,Y 0.000,Z 180.000,A 0.000,B 0.000,C 180.000,E1 0.000} C_DIS
LIN {X -228.480,Y -11.777,Z 180.000,A 0.000,B 0.000,C 180.000,E1 0.000} C_DIS
LIN {X -227.571,Y -23.524,Z 180.000,A 0.000,B 0.000,C 180.000,E1 0.000} C_DIS
LIN {X -226.059,Y -35.207,Z 180.000,A 0.000,B 0.000,C 180.000,E1 0.000} C_DIS
LIN {X -223.946,Y -46.798,Z 180.000,A 0.000,B 0.000,C 180.000,E1 0.000} C_DIS
LIN {X -221.240,Y -58.264,Z 180.000,A 0.000,B 0.000,C 180.000,E1 0.000} C_DIS
LIN {X -217.947,Y -69.576,Z 180.000,A 0.000,B 0.000,C 180.000,E1 0.000} C_DIS
LIN {X -214.077,Y -80.704,Z 180.000,A 0.000,B 0.000,C 180.000,E1 0.000} C_DIS
LIN {X -209.638,Y -91.618,Z 180.000,A 0.000,B 0.000,C 180.000,E1 0.000} C_DIS
LIN {X -204.645,Y -102.287,Z 180.000,A 0.000,B 0.000,C 180.000,E1 0.000} C_DIS
LIN {X -199.107,Y -112.687,Z 180.000,A 0.000,B 0.000,C 180.000,E1 0.000} C_DIS
LIN {X -193.042,Y -122.788,Z 180.000,A 0.000,B 0.000,C 180.000,E1 0.000} C_DIS
LIN {X -186.465,Y -132.562,Z 180.000,A 0.000,B 0.000,C 180.000,E1 0.000} C_DIS
LIN {X -179.393,Y -141.985,Z 180.000,A 0.000,B 0.000,C 180.000,E1 0.000} C_DIS
LIN {X -171.846,Y -151.032,Z 180.000,A 0.000,B 0.000,C 180.000,E1 0.000} C_DIS
LIN {X -163.844,Y -159.678,Z 180.000,A 0.000,B 0.000,C 180.000,E1 0.000} C_DIS
LIN {X -155.407,Y -167.901,Z 180.000,A 0.000,B 0.000,C 180.000,E1 0.000} C_DIS
LIN {X -146.558,Y -175.677,Z 180.000,A 0.000,B 0.000,C 180.000,E1 0.000} C_DIS
LIN {X -137.318,Y -182.990,Z 180.000,A 0.000,B 0.000,C 180.000,E1 0.000} C_DIS
LIN {X -127.717,Y -189.817,Z 180.000,A 0.000,B 0.000,C 180.000,E1 0.000} C_DIS
LIN {X -117.777,Y -196.140,Z 180.000,A 0.000,B 0.000,C 180.000,E1 0.000} C_DIS
LIN {X -107.524,Y -201.942,Z 180.000,A 0.000,B 0.000,C 180.000,E1 0.000} C_DIS
LIN {X -96.984,Y -207.209,Z 180.000,A 0.000,B 0.000,C 180.000,E1 0.000} C_DIS
LIN {X -86.189,Y -211.928,Z 180.000,A 0.000,B 0.000,C 180.000,E1 0.000} C_DIS
LIN {X -75.165,Y -216.084,Z 180.000,A 0.000,B 0.000,C 180.000,E1 0.000} C_DIS
LIN {X -63.942,Y -219.667,Z 180.000,A 0.000,B 0.000,C 180.000,E1 0.000} C_DIS
LIN {X -52.549,Y -222.667,Z 180.000,A 0.000,B 0.000,C 180.000,E1 0.000} C_DIS
LIN {X -41.016,Y -225.077,Z 180.000,A 0.000,B 0.000,C 180.000,E1 0.000} C_DIS
LIN {X -29.375,Y -226.890,Z 180.000,A 0.000,B 0.000,C 180.000,E1 0.000} C_DIS
LIN {X -17.657,Y -228.101,Z 180.000,A 0.000,B 0.000,C 180.000,E1 0.000} C_DIS
LIN {X -5.890,Y -228.708,Z 180.000,A 0.000,B 0.000,C 180.000,E1 0.000} C_DIS
LIN {X 5.890,Y -228.708,Z 180.000,A 0.000,B 0.000,C 180.000,E1 0.000} C_DIS
;rapid-leaky
$VEL.CP=0.3
LIN {X 5.490,Y -213.168,Z 180.000,A 0.000,B 0.000,C 180.000,E1 0.000} C_DIS
;bead-perimeter_inner
$VEL.CP=0.54
LIN {X 16.457,Y -212.603,Z 180.000,A 0.000,B 0.000,C 180.000,E1 0.000} C_DIS
LIN {X 27.379,Y -211.474,Z 180.000,A 0.000,B 0.000,C 180.000,E1 0.000} C_DIS
LIN {X 38.229,Y -209.784,Z 180.000,A 0.000,B 0.000,C 180.000,E1 0.000} C_DIS
LIN {X 48.978,Y -207.538,Z 180.000,A 0.000,B 0.000,C 180.000,E1 0.000} C_DIS
LIN {X 59.597,Y -204.741,Z 180.000,A 0.000,B 0.000,C 180.000,E1 0.000} C_DIS
LIN {X 70.057,Y -201.402,Z 180.000,A 0.000,B 0.000,C 180.000,E1 0.000} C_DIS
LIN {X 80.333,Y -197.527,Z 180.000,A 0.000,B 0.000,C 180.000,E1 0.000} C_DIS
LIN {X 90.392,Y -193.131,Z 180.000,A 0.000,B 0.000,C 180.000,E1 0.000} C_DIS
LIN {X 100.219,Y -188.220,Z 180.000,A 0.000,B 0.000,C 180.000,E1 0.000} C_DIS
LIN {X 109.775,Y -182.812,Z 180.000,A 0.000,B 0.000,C 180.000,E1 0.000} C_DIS
LIN {X 119.038,Y -176.920,Z 180.000,A 0.000,B 0.000,C 180.000,E1 0.000} C_DIS
LIN {X 127.988,Y -170.556,Z 180.000,A 0.000,B 0.000,C 180.000,E1 0.000} C_DIS
LIN {X 136.601,Y -163.740,Z 180.000,A 0.000,B 0.000,C 180.000,E1 0.000} C_DIS
LIN {X 144.847,Y -156.493,Z 180.000,A 0.000,B 0.000,C 180.000,E1 0.000} C_DIS
LIN {X 152.711,Y -148.829,Z 180.000,A 0.000,B 0.000,C 180.000,E1 0.000} C_DIS
LIN {X 160.170,Y -140.770,Z 180.000,A 0.000,B 0.000,C 180.000,E1 0.000} C_DIS
LIN {X 167.204,Y -132.337,Z 180.000,A 0.000,B 0.000,C 180.000,E1 0.000} C_DIS
LIN {X 173.796,Y -123.554,Z 180.000,A 0.000,B 0.000,C 180.000,E1 0.000} C_DIS
LIN {X 179.925,Y -114.445,Z 180.000,A 0.000,B 0.000,C 180.000,E1 0.000} C_DIS
LIN {X 185.578,Y -105.030,Z 180.000,A 0.000,B 0.000,C 180.000,E1 0.000} C_DIS
LIN {X 190.740,Y -95.337,Z 180.000,A 0.000,B 0.000,C 180.000,E1 0.000} C_DIS
LIN {X 195.394,Y -85.393,Z 180.000,A 0.000,B 0.000,C 180.000,E1 0.000} C_DIS
LIN {X 199.531,Y -75.221,Z 180.000,A 0.000,B 0.000,C 180.000,E1 0.000} C_DIS
LIN {X 203.138,Y -64.849,Z 180.000,A 0.000,B 0.000,C 180.000,E1 0.000} C_DIS
LIN {X 206.208,Y -54.305,Z 180.000,A 0.000,B 0.000,C 180.000,E1 0.000} C_DIS
LIN {X 208.730,Y -43.618,Z 180.000,A 0.000,B 0.000,C 180.000,E1 0.000} C_DIS
LIN {X 210.699,Y -32.815,Z 180.000,A 0.000,B 0.000,C 180.000,E1 0.000} C_DIS
LIN {X 212.108,Y -21.926,Z 180.000,A 0.000,B 0.000,C 180.000,E1 0.000} C_DIS
LIN {X 212.956,Y -10.977,Z 180.000,A 0.000,B 0.000,C 180.000,E1 0.000} C_DIS
LIN {X 213.239,Y 0.000,Z 180.000,A 0.000,B 0.000,C 180.000,E1 0.000} C_DIS
LIN {X 212.956,Y 10.977,Z 180.000,A 0.000,B 0.000,C 180.000,E1 0.000} C_DIS
LIN {X 212.108,Y 21.926,Z 180.000,A 0.000,B 0.000,C 180.000,E1 0.000} C_DIS
LIN {X 210.699,Y 32.815,Z 180.000,A 0.000,B 0.000,C 180.000,E1 0.000} C_DIS
LIN {X 208.730,Y 43.618,Z 180.000,A 0.000,B 0.000,C 180.000,E1 0.000} C_DIS
LIN {X 206.208,Y 54.305,Z 180.000,A 0.000,B 0.000,C 180.000,E1 0.000} C_DIS
LIN {X 203.138,Y 64.849,Z 180.000,A 0.000,B 0.000,C 180.000,E1 0.000} C_DIS
LIN {X 199.531,Y 75.221,Z 180.000,A 0.000,B 0.000,C 180.000,E1 0.000} C_DIS
LIN {X 195.394,Y 85.393,Z 180.000,A 0.000,B 0.000,C 180.000,E1 0.000} C_DIS
LIN {X 190.740,Y 95.337,Z 180.000,A 0.000,B 0.000,C 180.000,E1 0.000} C_DIS
LIN {X 185.578,Y 105.030,Z 180.000,A 0.000,B 0.000,C 180.000,E1 0.000} C_DIS
LIN {X 179.925,Y 114.445,Z 180.000,A 0.000,B 0.000,C 180.000,E1 0.000} C_DIS
LIN {X 173.796,Y 123.554,Z 180.000,A 0.000,B 0.000,C 180.000,E1 0.000} C_DIS
LIN {X 167.204,Y 132.337,Z 180.000,A 0.000,B 0.000,C 180.000,E1 0.000} C_DIS
LIN {X 160.170,Y 140.770,Z 180.000,A 0.000,B 0.000,C 180.000,E1 0.000} C_DIS
LIN {X 152.711,Y 148.829,Z 180.000,A 0.000,B 0.000,C 180.000,E1 0.000} C_DIS
LIN {X 144.847,Y 156.493,Z 180.000,A 0.000,B 0.000,C 180.000,E1 0.000} C_DIS
LIN {X 136.601,Y 163.740,Z 180.000,A 0.000,B 0.000,C 180.000,E1 0.000} C_DIS
LIN {X 127.988,Y 170.556,Z 180.000,A 0.000,B 0.000,C 180.000,E1 0.000} C_DIS
LIN {X 119.038,Y 176.920,Z 180.000,A 0.000,B 0.000,C 180.000,E1 0.000} C_DIS
LIN {X 109.775,Y 182.812,Z 180.000,A 0.000,B 0.000,C 180.000,E1 0.000} C_DIS
LIN {X 100.219,Y 188.220,Z 180.000,A 0.000,B 0.000,C 180.000,E1 0.000} C_DIS
LIN {X 90.394,Y 193.130,Z 180.000,A 0.000,B 0.000,C 180.000,E1 0.000} C_DIS
LIN {X 80.332,Y 197.528,Z 180.000,A 0.000,B 0.000,C 180.000,E1 0.000} C_DIS
LIN {X 70.057,Y 201.402,Z 180.000,A 0.000,B 0.000,C 180.000,E1 0.000} C_DIS
LIN {X 59.597,Y 204.741,Z 180.000,A 0.000,B 0.000,C 180.000,E1 0.000} C_DIS
LIN {X 48.978,Y 207.538,Z 180.000,A 0.000,B 0.000,C 180.000,E1 0.000} C_DIS
LIN {X 38.229,Y 209.784,Z 180.000,A 0.000,B 0.000,C 180.000,E1 0.000} C_DIS
LIN {X 27.379,Y 211.474,Z 180.000,A 0.000,B 0.000,C 180.000,E1 0.000} C_DIS
LIN {X 16.457,Y 212.603,Z 180.000,A 0.000,B 0.000,C 180.000,E1 0.000} C_DIS
LIN {X 5.490,Y 213.168,Z 180.000,A 0.000,B 0.000,C 180.000,E1 0.000} C_DIS
LIN {X -5.490,Y 213.168,Z 180.000,A 0.000,B 0.000,C 180.000,E1 0.000} C_DIS
LIN {X -16.457,Y 212.603,Z 180.000,A 0.000,B 0.000,C 180.000,E1 0.000} C_DIS
LIN {X -27.379,Y 211.474,Z 180.000,A 0.000,B 0.000,C 180.000,E1 0.000} C_DIS
LIN {X -38.229,Y 209.784,Z 180.000,A 0.000,B 0.000,C 180.000,E1 0.000} C_DIS
LIN {X -48.978,Y 207.538,Z 180.000,A 0.000,B 0.000,C 180.000,E1 0.000} C_DIS
LIN {X -59.597,Y 204.741,Z 180.000,A 0.000,B 0.000,C 180.000,E1 0.000} C_DIS
LIN {X -70.057,Y 201.402,Z 180.000,A 0.000,B 0.000,C 180.000,E1 0.000} C_DIS
LIN {X -80.333,Y 197.527,Z 180.000,A 0.000,B 0.000,C 180.000,E1 0.000} C_DIS
LIN {X -90.392,Y 193.131,Z 180.000,A 0.000,B 0.000,C 180.000,E1 0.000} C_DIS
LIN {X -100.219,Y 188.220,Z 180.000,A 0.000,B 0.000,C 180.000,E1 0.000} C_DIS
LIN {X -109.775,Y 182.812,Z 180.000,A 0.000,B 0.000,C 180.000,E1 0.000} C_DIS
LIN {X -119.038,Y 176.920,Z 180.000,A 0.000,B 0.000,C 180.000,E1 0.000} C_DIS
LIN {X -127.988,Y 170.556,Z 180.000,A 0.000,B 0.000,C 180.000,E1 0.000} C_DIS
LIN {X -136.601,Y 163.740,Z 180.000,A 0.000,B 0.000,C 180.000,E1 0.000} C_DIS
LIN {X -144.847,Y 156.493,Z 180.000,A 0.000,B 0.000,C 180.000,E1 0.000} C_DIS
LIN {X -152.711,Y 148.829,Z 180.000,A 0.000,B 0.000,C 180.000,E1 0.000} C_DIS
LIN {X -160.170,Y 140.770,Z 180.000,A 0.000,B 0.000,C 180.000,E1 0.000} C_DIS
LIN {X -167.204,Y 132.337,Z 180.000,A 0.000,B 0.000,C 180.000,E1 0.000} C_DIS
LIN {X -173.796,Y 123.554,Z 180.000,A 0.000,B 0.000,C 180.000,E1 0.000} C_DIS
LIN {X -179.925,Y 114.445,Z 180.000,A 0.000,B 0.000,C 180.000,E1 0.000} C_DIS
LIN {X -185.578,Y 105.030,Z 180.000,A 0.000,B 0.000,C 180.000,E1 0.000} C_DIS
LIN {X -190.740,Y 95.337,Z 180.000,A 0.000,B 0.000,C 180.000,E1 0.000} C_DIS
LIN {X -195.394,Y 85.393,Z 180.000,A 0.000,B 0.000,C 180.000,E1 0.000} C_DIS
LIN {X -199.531,Y 75.221,Z 180.000,A 0.000,B 0.000,C 180.000,E1 0.000} C_DIS
LIN {X -203.138,Y 64.849,Z 180.000,A 0.000,B 0.000,C 180.000,E1 0.000} C_DIS
LIN {X -206.208,Y 54.305,Z 180.000,A 0.000,B 0.000,C 180.000,E1 0.000} C_DIS
LIN {X -208.730,Y 43.618,Z 180.000,A 0.000,B 0.000,C 180.000,E1 0.000} C_DIS
LIN {X -210.699,Y 32.815,Z 180.000,A 0.000,B 0.000,C 180.000,E1 0.000} C_DIS
LIN {X -212.108,Y 21.926,Z 180.000,A 0.000,B 0.000,C 180.000,E1 0.000} C_DIS
LIN {X -212.956,Y 10.977,Z 180.000,A 0.000,B 0.000,C 180.000,E1 0.000} C_DIS
LIN {X -213.239,Y 0.000,Z 180.000,A 0.000,B 0.000,C 180.000,E1 0.000} C_DIS
LIN {X -212.956,Y -10.977,Z 180.000,A 0.000,B 0.000,C 180.000,E1 0.000} C_DIS
LIN {X -212.108,Y -21.926,Z 180.000,A 0.000,B 0.000,C 180.000,E1 0.000} C_DIS
LIN {X -210.699,Y -32.815,Z 180.000,A 0.000,B 0.000,C 180.000,E1 0.000} C_DIS
LIN {X -208.730,Y -43.618,Z 180.000,A 0.000,B 0.000,C 180.000,E1 0.000} C_DIS
LIN {X -206.208,Y -54.305,Z 180.000,A 0.000,B 0.000,C 180.000,E1 0.000} C_DIS
LIN {X -203.138,Y -64.849,Z 180.000,A 0.000,B 0.000,C 180.000,E1 0.000} C_DIS
LIN {X -199.531,Y -75.221,Z 180.000,A 0.000,B 0.000,C 180.000,E1 0.000} C_DIS
LIN {X -195.394,Y -85.393,Z 180.000,A 0.000,B 0.000,C 180.000,E1 0.000} C_DIS
LIN {X -190.740,Y -95.337,Z 180.000,A 0.000,B 0.000,C 180.000,E1 0.000} C_DIS
LIN {X -185.578,Y -105.030,Z 180.000,A 0.000,B 0.000,C 180.000,E1 0.000} C_DIS
LIN {X -179.925,Y -114.445,Z 180.000,A 0.000,B 0.000,C 180.000,E1 0.000} C_DIS
LIN {X -173.796,Y -123.554,Z 180.000,A 0.000,B 0.000,C 180.000,E1 0.000} C_DIS
LIN {X -167.204,Y -132.337,Z 180.000,A 0.000,B 0.000,C 180.000,E1 0.000} C_DIS
LIN {X -160.170,Y -140.770,Z 180.000,A 0.000,B 0.000,C 180.000,E1 0.000} C_DIS
LIN {X -152.711,Y -148.829,Z 180.000,A 0.000,B 0.000,C 180.000,E1 0.000} C_DIS
LIN {X -144.847,Y -156.493,Z 180.000,A 0.000,B 0.000,C 180.000,E1 0.000} C_DIS
LIN {X -136.601,Y -163.740,Z 180.000,A 0.000,B 0.000,C 180.000,E1 0.000} C_DIS
LIN {X -127.988,Y -170.556,Z 180.000,A 0.000,B 0.000,C 180.000,E1 0.000} C_DIS
LIN {X -119.038,Y -176.920,Z 180.000,A 0.000,B 0.000,C 180.000,E1 0.000} C_DIS
LIN {X -109.775,Y -182.812,Z 180.000,A 0.000,B 0.000,C 180.000,E1 0.000} C_DIS
LIN {X -100.219,Y -188.220,Z 180.000,A 0.000,B 0.000,C 180.000,E1 0.000} C_DIS
LIN {X -90.394,Y -193.130,Z 180.000,A 0.000,B 0.000,C 180.000,E1 0.000} C_DIS
LIN {X -80.332,Y -197.528,Z 180.000,A 0.000,B 0.000,C 180.000,E1 0.000} C_DIS
LIN {X -70.057,Y -201.402,Z 180.000,A 0.000,B 0.000,C 180.000,E1 0.000} C_DIS
LIN {X -59.597,Y -204.741,Z 180.000,A 0.000,B 0.000,C 180.000,E1 0.000} C_DIS
LIN {X -48.978,Y -207.538,Z 180.000,A 0.000,B 0.000,C 180.000,E1 0.000} C_DIS
LIN {X -38.229,Y -209.784,Z 180.000,A 0.000,B 0.000,C 180.000,E1 0.000} C_DIS
LIN {X -27.379,Y -211.474,Z 180.000,A 0.000,B 0.000,C 180.000,E1 0.000} C_DIS
LIN {X -16.457,Y -212.603,Z 180.000,A 0.000,B 0.000,C 180.000,E1 0.000} C_DIS
LIN {X -5.490,Y -213.168,Z 180.000,A 0.000,B 0.000,C 180.000,E1 0.000} C_DIS
LIN {X 5.490,Y -213.168,Z 180.000,A 0.000,B 0.000,C 180.000,E1 0.000} C_DIS
;rapid-leaky
$VEL.CP=0.3
LIN {X -195.295,Y -6.892,Z 180.000,A 0.000,B 0.000,C 180.000,E1 0.000} C_DIS
;bead-sparse_infill
$VEL.CP=0.54
LIN {X 6.908,Y 195.311,Z 180.000,A 0.000,B 0.000,C 180.000,E1 0.000} C_DIS
LIN {X 15.086,Y 194.890,Z 180.000,A 0.000,B 0.000,C 180.000,E1 0.000} C_DIS
LIN {X 25.098,Y 193.855,Z 180.000,A 0.000,B 0.000,C 180.000,E1 0.000} C_DIS
LIN {X 35.044,Y 192.306,Z 180.000,A 0.000,B 0.000,C 180.000,E1 0.000} C_DIS
LIN {X 44.897,Y 190.247,Z 180.000,A 0.000,B 0.000,C 180.000,E1 0.000} C_DIS
LIN {X 54.631,Y 187.683,Z 180.000,A 0.000,B 0.000,C 180.000,E1 0.000} C_DIS
LIN {X 64.220,Y 184.622,Z 180.000,A 0.000,B 0.000,C 180.000,E1 0.000} C_DIS
LIN {X 73.639,Y 181.071,Z 180.000,A 0.000,B 0.000,C 180.000,E1 0.000} C_DIS
LIN {X 82.863,Y 177.039,Z 180.000,A 0.000,B 0.000,C 180.000,E1 0.000} C_DIS
LIN {X 91.870,Y 172.538,Z 180.000,A 0.000,B 0.000,C 180.000,E1 0.000} C_DIS
LIN {X 100.629,Y 167.581,Z 180.000,A 0.000,B 0.000,C 180.000,E1 0.000} C_DIS
LIN {X 109.120,Y 162.180,Z 180.000,A 0.000,B 0.000,C 180.000,E1 0.000} C_DIS
LIN {X 117.324,Y 156.347,Z 180.000,A 0.000,B 0.000,C 180.000,E1 0.000} C_DIS
LIN {X 121.565,Y 152.991,Z 180.000,A 0.000,B 0.000,C 180.000,E1 0.000} C_DIS
LIN {X -153.030,Y -121.604,Z 180.000,A 0.000,B 0.000,C 180.000,E1 0.000} C_DIS
LIN {X -146.825,Y -129.042,Z 180.000,A 0.000,B 0.000,C 180.000,E1 0.000} C_DIS
LIN {X -139.988,Y -136.429,Z 180.000,A 0.000,B 0.000,C 180.000,E1 0.000} C_DIS
LIN {X -132.780,Y -143.454,Z 180.000,A 0.000,B 0.000,C 180.000,E1 0.000} C_DIS
LIN {X -125.220,Y -150.098,Z 180.000,A 0.000,B 0.000,C 180.000,E1 0.000} C_DIS
LIN {X -117.324,Y -156.347,Z 180.000,A 0.000,B 0.000,C 180.000,E1 0.000} C_DIS
LIN {X -109.120,Y -162.180,Z 180.000,A 0.000,B 0.000,C 180.000,E1 0.000} C_DIS
LIN {X -100.629,Y -167.581,Z 180.000,A 0.000,B 0.000,C 180.000,E1 0.000} C_DIS
LIN {X -91.870,Y -172.538,Z 180.000,A 0.000,B 0.000,C 180.000,E1 0.000} C_DIS
LIN {X -82.863,Y -177.039,Z 180.000,A 0.000,B 0.000,C 180.000,E1 0.000} C_DIS
LIN {X -73.639,Y -181.071,Z 180.000,A 0.000,B 0.000,C 180.000,E1 0.000} C_DIS
LIN {X -64.220,Y -184.622,Z 180.000,A 0.000,B 0.000,C 180.000,E1 0.000} C_DIS
LIN {X -60.316,Y -185.868,Z 180.000,A 0.000,B 0.000,C 180.000,E1 0.000} C_DIS
LIN {X 185.900,Y 60.348,Z 180.000,A 0.000,B 0.000,C 180.000,E1 0.000} C_DIS
;rapid-leaky
$VEL.CP=0.3
LIN {X -141.520,Y -169.640,Z 190.000,A 0.000,B 0.000,C 180.000,E1 0.000} C_DIS
;bead-perimeter_outer
$VEL.CP=0.52
LIN {X -132.599,Y -176.700,Z 190.000,A 0.000,B 0.000,C 180.000,E1 0.000} C_DIS
LIN {X -123.327,Y -183.292,Z 190.000,A 0.000,B 0.000,C 180.000,E1 0.000} C_DIS
LIN {X -113.728,Y -189.398,Z 190.000,A 0.000,B 0.000,C 180.000,E1 0.000} C_DIS
LIN {X -103.828,Y -195.001,Z 190.000,A 0.000,B 0.000,C 180.000,E1 0.000} C_DIS
LIN {X -93.651,Y -200.087,Z 190.000,A 0.000,B 0.000,C 180.000,E1 0.000} C_DIS
LIN {X -83.227,Y -204.643,Z 190.000,A 0.000,B 0.000,C 180.000,E1 0.000} C_DIS
LIN {X -72.581,Y -208.657,Z 190.000,A 0.000,B 0.000,C 180.000,E1 0.000} C_DIS
LIN {X -61.744,Y -212.116,Z 190.000,A 0.000,B 0.000,C 180.000,E1 0.000} C_DIS
LIN {X -50.743,Y -215.013,Z 190.000,A 0.000,B 0.000,C 180.000,E1 0.000} C_DIS
LIN {X -39.607,Y -217.340,Z 190.000,A 0.000,B 0.000,C 180.000,E1 0.000} C_DIS
LIN {X -28.365,Y -219.090,Z 190.000,A 0.000,B 0.000,C 180.000,E1 0.000} C_DIS
LIN {X -17.050,Y -220.260,Z 190.000,A 0.000,B 0.000,C 180.000,E1 0.000} C_DIS
LIN {X -5.688,Y -220.846,Z 190.000,A 0.000,B 0.000,C 180.000,E1 0.000} C_DIS
LIN {X 5.688,Y -220.846,Z 190.000,A 0.000,B 0.000,C 180.000,E1 0.000} C_DIS
LIN {X 17.050,Y -220.260,Z 190.000,A 0.000,B 0.000,C 180.000,E1 0.000} C_DIS
LIN {X 28.365,Y -219.090,Z 190.000,A 0.000,B 0.000,C 180.000,E1 0.000} C_DIS
LIN {X 39.607,Y -217.340,Z 190.000,A 0.000,B 0.000,C 180.000,E1 0.000} C_DIS
LIN {X 50.743,Y -215.013,Z 190.000,A 0.000,B 0.000,C 180.000,E1 0.000} C_DIS
LIN {X 61.744,Y -212.116,Z 190.000,A 0.000,B 0.000,C 180.000,E1 0.000} C_DIS
LIN {X 72.581,Y -208.657,Z 190.000,A 0.000,B 0.000,C 180.000,E1 0.000} C_DIS
LIN {X 83.227,Y -204.643,Z 190.000,A 0.000,B 0.000,C 180.000,E1 0.000} C_DIS
LIN {X 93.651,Y -200.087,Z 190.000,A 0.000,B 0.000,C 180.000,E1 0.000} C_DIS
LIN {X 103.828,Y -195.001,Z 190.000,A 0.000,B 0.000,C 180.000,E1 0.000} C_DIS
LIN {X 113.728,Y -189.398,Z 190.000,A 0.000,B 0.000,C 180.000,E1 0.000} C_DIS
LIN {X 123.327,Y -183.292,Z 190.000,A 0.000,B 0.000,C 180.000,E1 0.000} C_DIS
LIN {X 132.599,Y -176.700,Z 190.000,A 0.000,B 0.000,C 180.000,E1 0.000} C_DIS
LIN {X 141.520,Y -169.640,Z 190.000,A 0.000,B 0.000,C 180.000,E1 0.000} C_DIS
LIN {X 150.064,Y -162.129,Z 190.000,A 0.000,B 0.000,C 180.000,E1 0.000} C_DIS
LIN {X 158.212,Y -154.189,Z 190.000,A 0.000,B 0.000,C 180.000,E1 0.000} C_DIS
LIN {X 165.940,Y -145.841,Z 190.000,A 0.000,B 0.000,C 180.000,E1 0.000} C_DIS
LIN {X 173.227,Y -137.105,Z 190.000,A 0.000,B 0.000,C 180.000,E1 0.000} C_DIS
LIN {X 180.055,Y -128.005,Z 190.000,A 0.000,B 0.000,C 180.000,E1 0.000} C_DIS
LIN {X 186.406,Y -118.567,Z 190.000,A 0.000,B 0.000,C 180.000,E1 0.000} C_DIS
LIN {X 192.263,Y -108.813,Z 190.000,A 0.000,B 0.000,C 180.000,E1 0.000} C_DIS
LIN {X 197.610,Y -98.771,Z 190.000,A 0.000,B 0.000,C 180.000,E1 0.000} C_DIS
LIN {X 202.432,Y -88.468,Z 190.000,A 0.000,B 0.000,C 180.000,E1 0.000} C_DIS
LIN {X 206.718,Y -77.929,Z 190.000,A 0.000,B 0.000,C 180.000,E1 0.000} C_DIS
LIN {X 208.713,Y -72.196,Z 190.000,A 0.000,B 0.000,C 180.000,E1 0.000} C_DIS
LIN {X 210.455,Y -67.186,Z 190.000,A 0.000,B 0.000,C 180.000,E1 0.000} C_DIS
LIN {X 213.635,Y -56.261,Z 190.000,A 0.000,B 0.000,C 180.000,E1 0.000} C_DIS
LIN {X 216.248,Y -45.190,Z 190.000,A 0.000,B 0.000,C 180.000,E1 0.000} C_DIS
LIN {X 218.288,Y -33.997,Z 190.000,A 0.000,B 0.000,C 180.000,E1 0.000} C_DIS
LIN {X 219.748,Y -22.715,Z 190.000,A 0.000,B 0.000,C 180.000,E1 0.000} C_DIS
LIN {X 220.627,Y -11.372,Z 190.000,A 0.000,B 0.000,C 180.000,E1 0.000} C_DIS
LIN {X 220.919,Y 0.000,Z 190.000,A 0.000,B 0.000,C 180.000,E1 0.000} C_DIS
LIN {X 220.627,Y 11.372,Z 190.000,A 0.000,B 0.000,C 180.000,E1 0.000} C_DIS
LIN {X 219.748,Y 22.715,Z 190.000,A 0.000,B 0.000,C 180.000,E1 0.000} C_DIS
LIN {X 218.288,Y 33.997,Z 190.000,A 0.000,B 0.000,C 180.000,E1 0.000} C_DIS
LIN {X 216.248,Y 45.190,Z 190.000,A 0.000,B 0.000,C 180.000,E1 0.000} C_DIS
LIN {X 213.635,Y 56.261,Z 190.000,A 0.000,B 0.000,C 180.000,E1 0.000} C_DIS
LIN {X 210.455,Y 67.185,Z 190.000,A 0.000,B 0.000,C 180.000,E1 0.000} C_DIS
LIN {X 206.718,Y 77.929,Z 190.000,A 0.000,B 0.000,C 180.000,E1 0.000} C_DIS
LIN {X 202.432,Y 88.468,Z 190.000,A 0.000,B 0.000,C 180.000,E1 0.000} C_DIS
LIN {X 199.859,Y 93.967,Z 190.000,A 0.000,B 0.000,C 180.000,E1 0.000} C_DIS
LIN {X 197.610,Y 98.771,Z 190.000,A 0.000,B 0.000,C 180.000,E1 0.000} C_DIS
LIN {X 192.263,Y 108.813,Z 190.000,A 0.000,B 0.000,C 180.000,E1 0.000} C_DIS
LIN {X 186.406,Y 118.567,Z 190.000,A 0.000,B 0.000,C 180.000,E1 0.000} C_DIS
LIN {X 180.055,Y 128.005,Z 190.000,A 0.000,B 0.000,C 180.000,E1 0.000} C_DIS
LIN {X 173.227,Y 137.105,Z 190.000,A 0.000,B 0.000,C 180.000,E1 0.000} C_DIS
LIN {X 165.940,Y 145.841,Z 190.000,A 0.000,B 0.000,C 180.000,E1 0.000} C_DIS
LIN {X 158.212,Y 154.189,Z 190.000,A 0.000,B 0.000,C 180.000,E1 0.000} C_DIS
LIN {X 150.064,Y 162.129,Z 190.000,A 0.000,B 0.000,C 180.000,E1 0.000} C_DIS
LIN {X 141.520,Y 169.640,Z 190.000,A 0.000,B 0.000,C 180.000,E1 0.000} C_DIS
LIN {X 132.599,Y 176.700,Z 190.000,A 0.000,B 0.000,C 180.000,E1 0.000} C_DIS
LIN {X 123.327,Y 183.292,Z 190.000,A 0.000,B 0.000,C 180.000,E1 0.000} C_DIS
LIN {X 113.728,Y 189.398,Z 190.000,A 0.000,B 0.000,C 180.000,E1 0.000} C_DIS
LIN {X 103.828,Y 195.001,Z 190.000,A 0.000,B 0.000,C 180.000,E1 0.000} C_DIS
LIN {X 93.651,Y 200.087,Z 190.000,A 0.000,B 0.000,C 180.000,E1 0.000} C_DIS
LIN {X 83.227,Y 204.643,Z 190.000,A 0.000,B 0.000,C 180.000,E1 0.000} C_DIS
LIN {X 72.581,Y 208.657,Z 190.000,A 0.000,B 0.000,C 180.000,E1 0.000} C_DIS
LIN {X 61.744,Y 212.116,Z 190.000,A 0.000,B 0.000,C 180.000,E1 0.000} C_DIS
LIN {X 50.743,Y 215.013,Z 190.000,A 0.000,B 0.000,C 180.000,E1 0.000} C_DIS
LIN {X 39.607,Y 217.340,Z 190.000,A 0.000,B 0.000,C 180.000,E1 0.000} C_DIS
LIN {X 28.365,Y 219.090,Z 190.000,A 0.000,B 0.000,C 180.000,E1 0.000} C_DIS
LIN {X 17.050,Y 220.260,Z 190.000,A 0.000,B 0.000,C 180.000,E1 0.000} C_DIS
LIN {X 5.688,Y 220.846,Z 190.000,A 0.000,B 0.000,C 180.000,E1 0.000} C_DIS
LIN {X -5.688,Y 220.846,Z 190.000,A 0.000,B 0.000,C 180.000,E1 0.000} C_DIS
LIN {X -11.752,Y 220.534,Z 190.000,A 0.000,B 0.000,C 180.000,E1 0.000} C_DIS
LIN {X -17.050,Y 220.260,Z 190.000,A 0.000,B 0.000,C 180.000,E1 0.000} C_DIS
LIN {X -28.365,Y 219.090,Z 190.000,A 0.000,B 0.000,C 180.000,E1 0.000} C_DIS
LIN {X -39.607,Y 217.340,Z 190.000,A 0.000,B 0.000,C 180.000,E1 0.000} C_DIS
LIN {X -50.743,Y 215.013,Z 190.000,A 0.000,B 0.000,C 180.000,E1 0.000} C_DIS
LIN {X -61.744,Y 212.116,Z 190.000,A 0.000,B 0.000,C 180.000,E1 0.000} C_DIS
LIN {X -72.581,Y 208.657,Z 190.000,A 0.000,B 0.000,C 180.000,E1 0.000} C_DIS
LIN {X -83.227,Y 204.643,Z 190.000,A 0.000,B 0.000,C 180.000,E1 0.000} C_DIS
LIN {X -93.651,Y 200.087,Z 190.000,A 0.000,B 0.000,C 180.000,E1 0.000} C_DIS
LIN {X -103.828,Y 195.001,Z 190.000,A 0.000,B 0.000,C 180.000,E1 0.000} C_DIS
LIN {X -113.728,Y 189.398,Z 190.000,A 0.000,B 0.000,C 180.000,E1 0.000} C_DIS
LIN {X -123.327,Y 183.292,Z 190.000,A 0.000,B 0.000,C 180.000,E1 0.000} C_DIS
LIN {X -132.599,Y 176.700,Z 190.000,A 0.000,B 0.000,C 180.000,E1 0.000} C_DIS
LIN {X -141.520,Y 169.640,Z 190.000,A 0.000,B 0.000,C 180.000,E1 0.000} C_DIS
LIN {X -150.064,Y 162.129,Z 190.000,A 0.000,B 0.000,C 180.000,E1 0.000} C_DIS
LIN {X -158.212,Y 154.189,Z 190.000,A 0.000,B 0.000,C 180.000,E1 0.000} C_DIS
LIN {X -165.940,Y 145.841,Z 190.000,A 0.000,B 0.000,C 180.000,E1 0.000} C_DIS
LIN {X -173.227,Y 137.105,Z 190.000,A 0.000,B 0.000,C 180.000,E1 0.000} C_DIS
LIN {X -180.055,Y 128.005,Z 190.000,A 0.000,B 0.000,C 180.000,E1 0.000} C_DIS
LIN {X -186.406,Y 118.567,Z 190.000,A 0.000,B 0.000,C 180.000,E1 0.000} C_DIS
LIN {X -192.263,Y 108.813,Z 190.000,A 0.000,B 0.000,C 180.000,E1 0.000} C_DIS
LIN {X -197.610,Y 98.771,Z 190.000,A 0.000,B 0.000,C 180.000,E1 0.000} C_DIS
LIN {X -202.432,Y 88.468,Z 190.000,A 0.000,B 0.000,C 180.000,E1 0.000} C_DIS
LIN {X -206.718,Y 77.929,Z 190.000,A 0.000,B 0.000,C 180.000,E1 0.000} C_DIS
LIN {X -210.455,Y 67.186,Z 190.000,A 0.000,B 0.000,C 180.000,E1 0.000} C_DIS
LIN {X -213.635,Y 56.261,Z 190.000,A 0.000,B 0.000,C 180.000,E1 0.000} C_DIS
LIN {X -216.248,Y 45.190,Z 190.000,A 0.000,B 0.000,C 180.000,E1 0.000} C_DIS
LIN {X -218.288,Y 33.997,Z 190.000,A 0.000,B 0.000,C 180.000,E1 0.000} C_DIS
LIN {X -219.748,Y 22.715,Z 190.000,A 0.000,B 0.000,C 180.000,E1 0.000} C_DIS
LIN {X -220.627,Y 11.372,Z 190.000,A 0.000,B 0.000,C 180.000,E1 0.000} C_DIS
LIN {X -220.919,Y 0.000,Z 190.000,A 0.000,B 0.000,C 180.000,E1 0.000} C_DIS
LIN {X -220.627,Y -11.372,Z 190.000,A 0.000,B 0.000,C 180.000,E1 0.000} C_DIS
LIN {X -219.748,Y -22.715,Z 190.000,A 0.000,B 0.000,C 180.000,E1 0.000} C_DIS
LIN {X -218.288,Y -33.997,Z 190.000,A 0.000,B 0.000,C 180.000,E1 0.000} C_DIS
LIN {X -216.248,Y -45.190,Z 190.000,A 0.000,B 0.000,C 180.000,E1 0.000} C_DIS
LIN {X -213.635,Y -56.261,Z 190.000,A 0.000,B 0.000,C 180.000,E1 0.000} C_DIS
LIN {X -210.455,Y -67.185,Z 190.000,A 0.000,B 0.000,C 180.000,E1 0.000} C_DIS
LIN {X -206.718,Y -77.929,Z 190.000,A 0.000,B 0.000,C 180.000,E1 0.000} C_DIS
LIN {X -202.432,Y -88.468,Z 190.000,A 0.000,B 0.000,C 180.000,E1 0.000} C_DIS
LIN {X -197.610,Y -98.771,Z 190.000,A 0.000,B 0.000,C 180.000,E1 0.000} C_DIS
LIN {X -192.263,Y -108.813,Z 190.000,A 0.000,B 0.000,C 180.000,E1 0.000} C_DIS
LIN {X -186.406,Y -118.567,Z 190.000,A 0.000,B 0.000,C 180.000,E1 0.000} C_DIS
LIN {X -180.055,Y -128.005,Z 190.000,A 0.000,B 0.000,C 180.000,E1 0.000} C_DIS
LIN {X -173.227,Y -137.105,Z 190.000,A 0.000,B 0.000,C 180.000,E1 0.000} C_DIS
LIN {X -165.940,Y -145.841,Z 190.000,A 0.000,B 0.000,C 180.000,E1 0.000} C_DIS
LIN {X -158.212,Y -154.189,Z 190.000,A 0.000,B 0.000,C 180.000,E1 0.000} C_DIS
LIN {X -150.064,Y -162.129,Z 190.000,A 0.000,B 0.000,C 180.000,E1 0.000} C_DIS
LIN {X -141.520,Y -169.640,Z 190.000,A 0.000,B 0.000,C 180.000,E1 0.000} C_DIS
;rapid-leaky
$VEL.CP=0.3
LIN {X -131.562,Y -157.703,Z 190.000,A 0.000,B 0.000,C 180.000,E1 0.000} C_DIS
;bead-perimeter_inner
$VEL.CP=0.52
LIN {X -123.268,Y -164.266,Z 190.000,A 0.000,B 0.000,C 180.000,E1 0.000} C_DIS
LIN {X -114.649,Y -170.395,Z 190.000,A 0.000,B 0.000,C 180.000,E1 0.000} C_DIS
LIN {X -105.725,Y -176.071,Z 190.000,A 0.000,B 0.000,C 180.000,E1 0.000} C_DIS
LIN {X -96.522,Y -181.280,Z 190.000,A 0.000,B 0.000,C 180.000,E1 0.000} C_DIS
LIN {X -87.061,Y -186.008,Z 190.000,A 0.000,B 0.000,C 180.000,E1 0.000} C_DIS
LIN {X -77.370,Y -190.244,Z 190.000,A 0.000,B 0.000,C 180.000,E1 0.000} C_DIS
LIN {X -67.474,Y -193.974,Z 190.000,A 0.000,B 0.000,C 180.000,E1 0.000} C_DIS
LIN {X -57.399,Y -197.190,Z 190.000,A 0.000,B 0.000,C 180.000,E1 0.000} C_DIS
LIN {X -47.172,Y -199.884,Z 190.000,A 0.000,B 0.000,C 180.000,E1 0.000} C_DIS
LIN {X -36.820,Y -202.047,Z 190.000,A 0.000,B 0.000,C 180.000,E1 0.000} C_DIS
LIN {X -26.370,Y -203.674,Z 190.000,A 0.000,B 0.000,C 180.000,E1 0.000} C_DIS
LIN {X -15.850,Y -204.762,Z 190.000,A 0.000,B 0.000,C 180.000,E1 0.000} C_DIS
LIN {X -5.288,Y -205.306,Z 190.000,A 0.000,B 0.000,C 180.000,E1 0.000} C_DIS
LIN {X 5.288,Y -205.306,Z 190.000,A 0.000,B 0.000,C 180.000,E1 0.000} C_DIS
LIN {X 15.849,Y -204.762,Z 190.000,A 0.000,B 0.000,C 180.000,E1 0.000} C_DIS
LIN {X 26.370,Y -203.674,Z 190.000,A 0.000,B 0.000,C 180.000,E1 0.000} C_DIS
LIN {X 36.820,Y -202.047,Z 190.000,A 0.000,B 0.000,C 180.000,E1 0.000} C_DIS
LIN {X 47.172,Y -199.884,Z 190.000,A 0.000,B 0.000,C 180.000,E1 0.000} C_DIS
LIN {X 57.399,Y -197.190,Z 190.000,A 0.000,B 0.000,C 180.000,E1 0.000} C_DIS
LIN {X 67.474,Y -193.974,Z 190.000,A 0.000,B 0.000,C 180.000,E1 0.000} C_DIS
LIN {X 77.370,Y -190.244,Z 190.000,A 0.000,B 0.000,C 180.000,E1 0.000} C_DIS
LIN {X 87.061,Y -186.008,Z 190.000,A 0.000,B 0.000,C 180.000,E1 0.000} C_DIS
LIN {X 96.522,Y -181.280,Z 190.000,A 0.000,B 0.000,C 180.000,E1 0.000} C_DIS
LIN {X 105.725,Y -176.071,Z 190.000,A 0.000,B 0.000,C 180.000,E1 0.000} C_DIS
LIN {X 114.649,Y -170.395,Z 190.000,A 0.000,B 0.000,C 180.000,E1 0.000} C_DIS
LIN {X 123.268,Y -164.266,Z 190.000,A 0.000,B 0.000,C 180.000,E1 0.000} C_DIS
LIN {X 131.562,Y -157.703,Z 190.000,A 0.000,B 0.000,C 180.000,E1 0.000} C_DIS
LIN {X 139.505,Y -150.721,Z 190.000,A 0.000,B 0.000,C 180.000,E1 0.000} C_DIS
LIN {X 147.080,Y -143.339,Z 190.000,A 0.000,B 0.000,C 180.000,E1 0.000} C_DIS
LIN {X 154.263,Y -135.578,Z 190.000,A 0.000,B 0.000,C 180.000,E1 0.000} C_DIS
LIN {X 161.038,Y -127.458,Z 190.000,A 0.000,B 0.000,C 180.000,E1 0.000} C_DIS
LIN {X 167.385,Y -118.999,Z 190.000,A 0.000,B 0.000,C 180.000,E1 0.000} C_DIS
LIN {X 173.289,Y -110.224,Z 190.000,A 0.000,B 0.000,C 180.000,E1 0.000} C_DIS
LIN {X 178.734,Y -101.156,Z 190.000,A 0.000,B 0.000,C 180.000,E1 0.000} C_DIS
LIN {X 183.705,Y -91.821,Z 190.000,A 0.000,B 0.000,C 180.000,E1 0.000} C_DIS
LIN {X 188.188,Y -82.243,Z 190.000,A 0.000,B 0.000,C 180.000,E1 0.000} C_DIS
LIN {X 192.173,Y -72.445,Z 190.000,A 0.000,B 0.000,C 180.000,E1 0.000} C_DIS
LIN {X 194.035,Y -67.092,Z 190.000,A 0.000,B 0.000,C 180.000,E1 0.000} C_DIS
LIN {X 195.646,Y -62.459,Z 190.000,A 0.000,B 0.000,C 180.000,E1 0.000} C_DIS
LIN {X 198.603,Y -52.302,Z 190.000,A 0.000,B 0.000,C 180.000,E1 0.000} C_DIS
LIN {X 201.032,Y -42.010,Z 190.000,A 0.000,B 0.000,C 180.000,E1 0.000} C_DIS
LIN {X 202.928,Y -31.605,Z 190.000,A 0.000,B 0.000,C 180.000,E1 0.000} C_DIS
LIN {X 204.286,Y -21.116,Z 190.000,A 0.000,B 0.000,C 180.000,E1 0.000} C_DIS
LIN {X 205.102,Y -10.572,Z 190.000,A 0.000,B 0.000,C 180.000,E1 0.000} C_DIS
LIN {X 205.374,Y 0.000,Z 190.000,A 0.000,B 0.000,C 180.000,E1 0.000} C_DIS
LIN {X 205.102,Y 10.572,Z 190.000,A 0.000,B 0.000,C 180.000,E1 0.000} C_DIS
LIN {X 204.286,Y 21.116,Z 190.000,A 0.000,B 0.000,C 180.000,E1 0.000} C_DIS
LIN {X 202.928,Y 31.605,Z 190.000,A 0.000,B 0.000,C 180.000,E1 0.000} C_DIS
LIN {X 201.032,Y 42.010,Z 190.000,A 0.000,B 0.000,C 180.000,E1 0.000} C_DIS
LIN {X 198.603,Y 52.302,Z 190.000,A 0.000,B 0.000,C 180.000,E1 0.000} C_DIS
LIN {X 195.646,Y 62.457,Z 190.000,A 0.000,B 0.000,C 180.000,E1 0.000} C_DIS
LIN {X 192.172,Y 72.446,Z 190.000,A 0.000,B 0.000,C 180.000,E1 0.000} C_DIS
LIN {X 188.188,Y 82.243,Z 190.000,A 0.000,B 0.000,C 180.000,E1 0.000} C_DIS
LIN {X 185.785,Y 87.379,Z 190.000,A 0.000,B 0.000,C 180.000,E1 0.000} C_DIS
LIN {X 183.706,Y 91.820,Z 190.000,A 0.000,B 0.000,C 180.000,E1 0.000} C_DIS
LIN {X 178.734,Y 101.156,Z 190.000,A 0.000,B 0.000,C 180.000,E1 0.000} C_DIS
LIN {X 173.289,Y 110.224,Z 190.000,A 0.000,B 0.000,C 180.000,E1 0.000} C_DIS
LIN {X 167.385,Y 118.999,Z 190.000,A 0.000,B 0.000,C 180.000,E1 0.000} C_DIS
LIN {X 161.038,Y 127.458,Z 190.000,A 0.000,B 0.000,C 180.000,E1 0.000} C_DIS
LIN {X 154.263,Y 135.578,Z 190.000,A 0.000,B 0.000,C 180.000,E1 0.000} C_DIS
LIN {X 147.080,Y 143.339,Z 190.000,A 0.000,B 0.000,C 180.000,E1 0.000} C_DIS
LIN {X 139.505,Y 150.721,Z 190.000,A 0.000,B 0.000,C 180.000,E1 0.000} C_DIS
LIN {X 131.562,Y 157.703,Z 190.000,A 0.000,B 0.000,C 180.000,E1 0.000} C_DIS
LIN {X 123.268,Y 164.266,Z 190.000,A 0.000,B 0.000,C 180.000,E1 0.000} C_DIS
LIN {X 114.649,Y 170.395,Z 190.000,A 0.000,B 0.000,C 180.000,E1 0.000} C_DIS
LIN {X 105.725,Y 176.071,Z 190.000,A 0.000,B 0.000,C 180.000,E1 0.000} C_DIS
LIN {X 96.522,Y 181.280,Z 190.000,A 0.000,B 0.000,C 180.000,E1 0.000} C_DIS
LIN {X 87.061,Y 186.008,Z 190.000,A 0.000,B 0.000,C 180.000,E1 0.000} C_DIS
LIN {X 77.370,Y 190.244,Z 190.000,A 0.000,B 0.000,C 180.000,E1 0.000} C_DIS
LIN {X 67.474,Y 193.974,Z 190.000,A 0.000,B 0.000,C 180.000,E1 0.000} C_DIS
LIN {X 57.399,Y 197.190,Z 190.000,A 0.000,B 0.000,C 180.000,E1 0.000} C_DIS
LIN {X 47.172,Y 199.884,Z 190.000,A 0.000,B 0.000,C 180.000,E1 0.000} C_DIS
LIN {X 36.820,Y 202.047,Z 190.000,A 0.000,B 0.000,C 180.000,E1 0.000} C_DIS
LIN {X 26.370,Y 203.674,Z 190.000,A 0.000,B 0.000,C 180.000,E1 0.000} C_DIS
LIN {X 15.850,Y 204.762,Z 190.000,A 0.000,B 0.000,C 180.000,E1 0.000} C_DIS
LIN {X 5.288,Y 205.306,Z 190.000,A 0.000,B 0.000,C 180.000,E1 0.000} C_DIS
LIN {X -5.288,Y 205.306,Z 190.000,A 0.000,B 0.000,C 180.000,E1 0.000} C_DIS
LIN {X -10.952,Y 205.014,Z 190.000,A 0.000,B 0.000,C 180.000,E1 0.000} C_DIS
LIN {X -15.849,Y 204.762,Z 190.000,A 0.000,B 0.000,C 180.000,E1 0.000} C_DIS
LIN {X -26.370,Y 203.674,Z 190.000,A 0.000,B 0.000,C 180.000,E1 0.000} C_DIS
LIN {X -36.820,Y 202.047,Z 190.000,A 0.000,B 0.000,C 180.000,E1 0.000} C_DIS
LIN {X -47.172,Y 199.884,Z 190.000,A 0.000,B 0.000,C 180.000,E1 0.000} C_DIS
LIN {X -57.399,Y 197.190,Z 190.000,A 0.000,B 0.000,C 180.000,E1 0.000} C_DIS
LIN {X -67.474,Y 193.974,Z 190.000,A 0.000,B 0.000,C 180.000,E1 0.000} C_DIS
LIN {X -77.370,Y 190.244,Z 190.000,A 0.000,B 0.000,C 180.000,E1 0.000} C_DIS
LIN {X -87.061,Y 186.008,Z 190.000,A 0.000,B 0.000,C 180.000,E1 0.000} C_DIS
LIN {X -96.522,Y 181.280,Z 190.000,A 0.000,B 0.000,C 180.000,E1 0.000} C_DIS
LIN {X -105.725,Y 176.071,Z 190.000,A 0.000,B 0.000,C 180.000,E1 0.000} C_DIS
LIN {X -114.649,Y 170.395,Z 190.000,A 0.000,B 0.000,C 180.000,E1 0.000} C_DIS
LIN {X -123.268,Y 164.266,Z 190.000,A 0.000,B 0.000,C 180.000,E1 0.000} C_DIS
LIN {X -131.562,Y 157.703,Z 190.000,A 0.000,B 0.000,C 180.000,E1 0.000} C_DIS
LIN {X -139.505,Y 150.721,Z 190.000,A 0.000,B 0.000,C 180.000,E1 0.000} C_DIS
LIN {X -147.080,Y 143.339,Z 190.000,A 0.000,B 0.000,C 180.000,E1 0.000} C_DIS
LIN {X -154.263,Y 135.578,Z 190.000,A 0.000,B 0.000,C 180.000,E1 0.000} C_DIS
LIN {X -161.038,Y 127.458,Z 190.000,A 0.000,B 0.000,C 180.000,E1 0.000} C_DIS
LIN {X -167.385,Y 118.999,Z 190.000,A 0.000,B 0.000,C 180.000,E1 0.000} C_DIS
LIN {X -173.289,Y 110.224,Z 190.000,A 0.000,B 0.000,C 180.000,E1 0.000} C_DIS
LIN {X -178.734,Y 101.156,Z 190.000,A 0.000,B 0.000,C 180.000,E1 0.000} C_DIS
LIN {X -183.705,Y 91.821,Z 190.000,A 0.000,B 0.000,C 180.000,E1 0.000} C_DIS
LIN {X -188.188,Y 82.243,Z 190.000,A 0.000,B 0.000,C 180.000,E1 0.000} C_DIS
LIN {X -192.173,Y 72.445,Z 190.000,A 0.000,B 0.000,C 180.000,E1 0.000} C_DIS
LIN {X -195.646,Y 62.459,Z 190.000,A 0.000,B 0.000,C 180.000,E1 0.000} C_DIS
LIN {X -198.603,Y 52.302,Z 190.000,A 0.000,B 0.000,C 180.000,E1 0.000} C_DIS
LIN {X -201.032,Y 42.010,Z 190.000,A 0.000,B 0.000,C 180.000,E1 0.000} C_DIS
LIN {X -202.928,Y 31.605,Z 190.000,A 0.000,B 0.000,C 180.000,E1 0.000} C_DIS
LIN {X -204.286,Y 21.116,Z 190.000,A 0.000,B 0.000,C 180.000,E1 0.000} C_DIS
LIN {X -205.102,Y 10.572,Z 190.000,A 0.000,B 0.000,C 180.000,E1 0.000} C_DIS
LIN {X -205.374,Y 0.000,Z 190.000,A 0.000,B 0.000,C 180.000,E1 0.000} C_DIS
LIN {X -205.102,Y -10.572,Z 190.000,A 0.000,B 0.000,C 180.000,E1 0.000} C_DIS
LIN {X -204.286,Y -21.116,Z 190.000,A 0.000,B 0.000,C 180.000,E1 0.000} C_DIS
LIN {X -202.928,Y -31.605,Z 190.000,A 0.000,B 0.000,C 180.000,E1 0.000} C_DIS
LIN {X -201.032,Y -42.010,Z 190.000,A 0.000,B 0.000,C 180.000,E1 0.000} C_DIS
LIN {X -198.603,Y -52.302,Z 190.000,A 0.000,B 0.000,C 180.000,E1 0.000} C_DIS
LIN {X -195.646,Y -62.457,Z 190.000,A 0.000,B 0.000,C 180.000,E1 0.000} C_DIS
LIN {X -192.172,Y -72.446,Z 190.000,A 0.000,B 0.000,C 180.000,E1 0.000} C_DIS
LIN {X -188.188,Y -82.243,Z 190.000,A 0.000,B 0.000,C 180.000,E1 0.000} C_DIS
LIN {X -183.706,Y -91.820,Z 190.000,A 0.000,B 0.000,C 180.000,E1 0.000} C_DIS
LIN {X -178.734,Y -101.156,Z 190.000,A 0.000,B 0.000,C 180.000,E1 0.000} C_DIS
LIN {X -173.289,Y -110.224,Z 190.000,A 0.000,B 0.000,C 180.000,E1 0.000} C_DIS
LIN {X -167.385,Y -118.999,Z 190.000,A 0.000,B 0.000,C 180.000,E1 0.000} C_DIS
LIN {X -161.038,Y -127.458,Z 190.000,A 0.000,B 0.000,C 180.000,E1 0.000} C_DIS
LIN {X -154.263,Y -135.578,Z 190.000,A 0.000,B 0.000,C 180.000,E1 0.000} C_DIS
LIN {X -147.080,Y -143.339,Z 190.000,A 0.000,B 0.000,C 180.000,E1 0.000} C_DIS
LIN {X -139.505,Y -150.721,Z 190.000,A 0.000,B 0.000,C 180.000,E1 0.000} C_DIS
LIN {X -131.562,Y -157.703,Z 190.000,A 0.000,B 0.000,C 180.000,E1 0.000} C_DIS
;rapid-leaky
$VEL.CP=0.3
LIN {X -0.857,Y -187.546,Z 190.000,A 0.000,B 0.000,C 180.000,E1 0.000} C_DIS
;bead-sparse_infill
$VEL.CP=0.52
LIN {X -187.587,Y -0.816,Z 190.000,A 0.000,B 0.000,C 180.000,E1 0.000} C_DIS
LIN {X -187.608,Y 0.000,Z 190.000,A 0.000,B 0.000,C 180.000,E1 0.000} C_DIS
LIN {X -187.360,Y 9.657,Z 190.000,A 0.000,B 0.000,C 180.000,E1 0.000} C_DIS
LIN {X -186.614,Y 19.289,Z 190.000,A 0.000,B 0.000,C 180.000,E1 0.000} C_DIS
LIN {X -185.373,Y 28.871,Z 190.000,A 0.000,B 0.000,C 180.000,E1 0.000} C_DIS
LIN {X -183.641,Y 38.376,Z 190.000,A 0.000,B 0.000,C 180.000,E1 0.000} C_DIS
LIN {X -181.423,Y 47.778,Z 190.000,A 0.000,B 0.000,C 180.000,E1 0.000} C_DIS
LIN {X -178.722,Y 57.056,Z 190.000,A 0.000,B 0.000,C 180.000,E1 0.000} C_DIS
LIN {X -175.549,Y 66.178,Z 190.000,A 0.000,B 0.000,C 180.000,E1 0.000} C_DIS
LIN {X -171.909,Y 75.129,Z 190.000,A 0.000,B 0.000,C 180.000,E1 0.000} C_DIS
LIN {X -167.814,Y 83.878,Z 190.000,A 0.000,B 0.000,C 180.000,E1 0.000} C_DIS
LIN {X -163.273,Y 92.405,Z 190.000,A 0.000,B 0.000,C 180.000,E1 0.000} C_DIS
LIN {X -158.299,Y 100.689,Z 190.000,A 0.000,B 0.000,C 180.000,E1 0.000} C_DIS
LIN {X -152.905,Y 108.705,Z 190.000,A 0.000,B 0.000,C 180.000,E1 0.000} C_DIS
LIN {X -147.429,Y 116.003,Z 190.000,A 0.000,B 0.000,C 180.000,E1 0.000} C_DIS
LIN {X 115.969,Y -147.394,Z 190.000,A 0.000,B 0.000,C 180.000,E1 0.000} C_DIS
LIN {X 120.181,Y -144.061,Z 190.000,A 0.000,B 0.000,C 180.000,E1 0.000} C_DIS
LIN {X 127.437,Y -137.683,Z 190.000,A 0.000,B 0.000,C 180.000,E1 0.000} C_DIS
LIN {X 134.357,Y -130.939,Z 190.000,A 0.000,B 0.000,C 180.000,E1 0.000} C_DIS
LIN {X 140.919,Y -123.850,Z 190.000,A 0.000,B 0.000,C 180.000,E1 0.000} C_DIS
LIN {X 147.107,Y -116.433,Z 190.000,A 0.000,B 0.000,C 180.000,E1 0.000} C_DIS
LIN {X 152.905,Y -108.705,Z 190.000,A 0.000,B 0.000,C 180.000,E1 0.000} C_DIS
LIN {X 158.299,Y -100.689,Z 190.000,A 0.000,B 0.000,C 180.000,E1 0.000} C_DIS
LIN {X 163.273,Y -92.405,Z 190.000,A 0.000,B 0.000,C 180.000,E1 0.000} C_DIS
LIN {X 167.814,Y -83.878,Z 190.000,A 0.000,B 0.000,C 180.000,E1 0.000} C_DIS
LIN {X 171.909,Y -75.129,Z 190.000,A 0.000,B 0.000,C 180.000,E1 0.000} C_DIS
LIN {X 175.549,Y -66.178,Z 190.000,A 0.000,B 0.000,C 180.000,E1 0.000} C_DIS
LIN {X 177.259,Y -61.261,Z 190.000,A 0.000,B 0.000,C 180.000,E1 0.000} C_DIS
LIN {X 178.722,Y -57.056,Z 190.000,A 0.000,B 0.000,C 180.000,E1 0.000} C_DIS
LIN {X 179.598,Y -54.046,Z 190.000,A 0.000,B 0.000,C 180.000,E1 0.000} C_DIS
LIN {X -54.061,Y 179.613,Z 190.000,A 0.000,B 0.000,C 180.000,E1 0.000} C_DIS
;rapid-leaky
$VEL.CP=0.3
LIN {X 38.075,Y -208.934,Z 200.000,A 0.000,B 0.000,C 180.000,E1 0.000} C_DIS
;bead-perimeter_outer
$VEL.CP=0.49
LIN {X 48.780,Y -206.698,Z 200.000,A 0.000,B 0.000,C 180.000,E1 0.000} C_DIS
LIN {X 59.356,Y -203.913,Z 200.000,A 0.000,B 0.000,C 180.000,E1 0.000} C_DIS
LIN {X 69.774,Y -200.587,Z 200.000,A 0.000,B 0.000,C 180.000,E1 0.000} C_DIS
LIN {X 80.008,Y -196.729,Z 200.000,A 0.000,B 0.000,C 180.000,E1 0.000} C_DIS
LIN {X 90.029,Y -192.349,Z 200.000,A 0.000,B 0.000,C 180.000,E1 0.000} C_DIS
LIN {X 99.811,Y -187.460,Z 200.000,A 0.000,B 0.000,C 180.000,E1 0.000} C_DIS
LIN {X 109.329,Y -182.073,Z 200.000,A 0.000,B 0.000,C 180.000,E1 0.000} C_DIS
LIN {X 118.557,Y -176.204,Z 200.000,A 0.000,B 0.000,C 180.000,E1 0.000} C_DIS
LIN {X 127.471,Y -169.866,Z 200.000,A 0.000,B 0.000,C 180.000,E1 0.000} C_DIS
LIN {X 136.047,Y -163.079,Z 200.000,A 0.000,B 0.000,C 180.000,E1 0.000} C_DIS
LIN {X 144.261,Y -155.859,Z 200.000,A 0.000,B 0.000,C 180.000,E1 0.000} C_DIS
LIN {X 152.094,Y -148.226,Z 200.000,A 0.000,B 0.000,C 180.000,E1 0.000} C_DIS
LIN {X 159.522,Y -140.201,Z 200.000,A 0.000,B 0.000,C 180.000,E1 0.000} C_DIS
LIN {X 166.527,Y -131.803,Z 200.000,A 0.000,B 0.000,C 180.000,E1 0.000} C_DIS
LIN {X 173.092,Y -123.055,Z 200.000,A 0.000,B 0.000,C 180.000,E1 0.000} C_DIS
LIN {X 179.197,Y -113.982,Z 200.000,A 0.000,B 0.000,C 180.000,E1 0.000} C_DIS
LIN {X 184.828,Y -104.605,Z 200.000,A 0.000,B 0.000,C 180.000,E1 0.000} C_DIS
LIN {X 189.967,Y -94.952,Z 200.000,A 0.000,B 0.000,C 180.000,E1 0.000} C_DIS
LIN {X 194.604,Y -85.046,Z 200.000,A 0.000,B 0.000,C 180.000,E1 0.000} C_DIS
LIN {X 198.724,Y -74.916,Z 200.000,A 0.000,B 0.000,C 180.000,E1 0.000} C_DIS
LIN {X 202.316,Y -64.586,Z 200.000,A 0.000,B 0.000,C 180.000,E1 0.000} C_DIS
LIN {X 205.373,Y -54.086,Z 200.000,A 0.000,B 0.000,C 180.000,E1 0.000} C_DIS
LIN {X 207.885,Y -43.441,Z 200.000,A 0.000,B 0.000,C 180.000,E1 0.000} C_DIS
LIN {X 209.847,Y -32.683,Z 200.000,A 0.000,B 0.000,C 180.000,E1 0.000} C_DIS
LIN {X 211.250,Y -21.836,Z 200.000,A 0.000,B 0.000,C 180.000,E1 0.000} C_DIS
LIN {X 212.095,Y -10.933,Z 200.000,A 0.000,B 0.000,C 180.000,E1 0.000} C_DIS
LIN {X 212.375,Y 0.000,Z 200.000,A 0.000,B 0.000,C 180.000,E1 0.000} C_DIS
LIN {X 212.095,Y 10.933,Z 200.000,A 0.000,B 0.000,C 180.000,E1 0.000} C_DIS
LIN {X 211.250,Y 21.836,Z 200.000,A 0.000,B 0.000,C 180.000,E1 0.000} C_DIS
LIN {X 209.847,Y 32.683,Z 200.000,A 0.000,B 0.000,C 180.000,E1 0.000} C_DIS
LIN {X 207.885,Y 43.441,Z 200.000,A 0.000,B 0.000,C 180.000,E1 0.000} C_DIS
LIN {X 205.373,Y 54.086,Z 200.000,A 0.000,B 0.000,C 180.000,E1 0.000} C_DIS
LIN {X 202.316,Y 64.586,Z 200.000,A 0.000,B 0.000,C 180.000,E1 0.000} C_DIS
LIN {X 198.724,Y 74.916,Z 200.000,A 0.000,B 0.000,C 180.000,E1 0.000} C_DIS
LIN {X 194.604,Y 85.046,Z 200.000,A 0.000,B 0.000,C 180.000,E1 0.000} C_DIS
LIN {X 192.793,Y 88.915,Z 200.000,A 0.000,B 0.000,C 180.000,E1 0.000} C_DIS
LIN {X 189.967,Y 94.951,Z 200.000,A 0.000,B 0.000,C 180.000,E1 0.000} C_DIS
LIN {X 184.828,Y 104.605,Z 200.000,A 0.000,B 0.000,C 180.000,E1 0.000} C_DIS
LIN {X 179.197,Y 113.982,Z 200.000,A 0.000,B 0.000,C 180.000,E1 0.000} C_DIS
LIN {X 173.092,Y 123.055,Z 200.000,A 0.000,B 0.000,C 180.000,E1 0.000} C_DIS
LIN {X 166.527,Y 131.803,Z 200.000,A 0.000,B 0.000,C 180.000,E1 0.000} C_DIS
LIN {X 159.522,Y 140.201,Z 200.000,A 0.000,B 0.000,C 180.000,E1 0.000} C_DIS
LIN {X 152.094,Y 148.226,Z 200.000,A 0.000,B 0.000,C 180.000,E1 0.000} C_DIS
LIN {X 144.261,Y 155.859,Z 200.000,A 0.000,B 0.000,C 180.000,E1 0.000} C_DIS
LIN {X 136.047,Y 163.079,Z 200.000,A 0.000,B 0.000,C 180.000,E1 0.000} C_DIS
LIN {X 127.471,Y 169.866,Z 200.000,A 0.000,B 0.000,C 180.000,E1 0.000} C_DIS
LIN {X 118.557,Y 176.204,Z 200.000,A 0.000,B 0.000,C 180.000,E1 0.000} C_DIS
LIN {X 109.329,Y 182.073,Z 200.000,A 0.000,B 0.000,C 180.000,E1 0.000} C_DIS
LIN {X 99.811,Y 187.460,Z 200.000,A 0.000,B 0.000,C 180.000,E1 0.000} C_DIS
LIN {X 90.029,Y 192.349,Z 200.000,A 0.000,B 0.000,C 180.000,E1 0.000} C_DIS
LIN {X 80.008,Y 196.730,Z 200.000,A 0.000,B 0.000,C 180.000,E1 0.000} C_DIS
LIN {X 76.010,Y 198.237,Z 200.000,A 0.000,B 0.000,C 180.000,E1 0.000} C_DIS
LIN {X 69.774,Y 200.587,Z 200.000,A 0.000,B 0.000,C 180.000,E1 0.000} C_DIS
LIN {X 59.356,Y 203.913,Z 200.000,A 0.000,B 0.000,C 180.000,E1 0.000} C_DIS
LIN {X 48.780,Y 206.698,Z 200.000,A 0.000,B 0.000,C 180.000,E1 0.000} C_DIS
LIN {X 38.075,Y 208.934,Z 200.000,A 0.000,B 0.000,C 180.000,E1 0.000} C_DIS
LIN {X 27.269,Y 210.617,Z 200.000,A 0.000,B 0.000,C 180.000,E1 0.000} C_DIS
LIN {X 16.389,Y 211.742,Z 200.000,A 0.000,B 0.000,C 180.000,E1 0.000} C_DIS
LIN {X 5.468,Y 212.306,Z 200.000,A 0.000,B 0.000,C 180.000,E1 0.000} C_DIS
LIN {X -5.468,Y 212.306,Z 200.000,A 0.000,B 0.000,C 180.000,E1 0.000} C_DIS
LIN {X -16.389,Y 211.742,Z 200.000,A 0.000,B 0.000,C 180.000,E1 0.000} C_DIS
LIN {X -27.269,Y 210.617,Z 200.000,A 0.000,B 0.000,C 180.000,E1 0.000} C_DIS
LIN {X -38.075,Y 208.934,Z 200.000,A 0.000,B 0.000,C 180.000,E1 0.000} C_DIS
LIN {X -48.780,Y 206.698,Z 200.000,A 0.000,B 0.000,C 180.000,E1 0.000} C_DIS
LIN {X -59.356,Y 203.913,Z 200.000,A 0.000,B 0.000,C 180.000,E1 0.000} C_DIS
LIN {X -69.774,Y 200.587,Z 200.000,A 0.000,B 0.000,C 180.000,E1 0.000} C_DIS
LIN {X -80.008,Y 196.729,Z 200.000,A 0.000,B 0.000,C 180.000,E1 0.000} C_DIS
LIN {X -90.029,Y 192.349,Z 200.000,A 0.000,B 0.000,C 180.000,E1 0.000} C_DIS
LIN {X -99.811,Y 187.460,Z 200.000,A 0.000,B 0.000,C 180.000,E1 0.000} C_DIS
LIN {X -109.329,Y 182.073,Z 200.000,A 0.000,B 0.000,C 180.000,E1 0.000} C_DIS
LIN {X -118.557,Y 176.204,Z 200.000,A 0.000,B 0.000,C 180.000,E1 0.000} C_DIS
LIN {X -127.471,Y 169.866,Z 200.000,A 0.000,B 0.000,C 180.000,E1 0.000} C_DIS
LIN {X -136.047,Y 163.079,Z 200.000,A 0.000,B 0.000,C 180.000,E1 0.000} C_DIS
LIN {X -144.261,Y 155.859,Z 200.000,A 0.000,B 0.000,C 180.000,E1 0.000} C_DIS
LIN {X -152.094,Y 148.226,Z 200.000,A 0.000,B 0.000,C 180.000,E1 0.000} C_DIS
LIN {X -159.522,Y 140.201,Z 200.000,A 0.000,B 0.000,C 180.000,E1 0.000} C_DIS
LIN {X -166.527,Y 131.803,Z 200.000,A 0.000,B 0.000,C 180.000,E1 0.000} C_DIS
LIN {X -173.092,Y 123.055,Z 200.000,A 0.000,B 0.000,C 180.000,E1 0.000} C_DIS
LIN {X -179.197,Y 113.982,Z 200.000,A 0.000,B 0.000,C 180.000,E1 0.000} C_DIS
LIN {X -184.828,Y 104.605,Z 200.000,A 0.000,B 0.000,C 180.000,E1 0.000} C_DIS
LIN {X -189.967,Y 94.952,Z 200.000,A 0.000,B 0.000,C 180.000,E1 0.000} C_DIS
LIN {X -194.604,Y 85.046,Z 200.000,A 0.000,B 0.000,C 180.000,E1 0.000} C_DIS
LIN {X -198.724,Y 74.916,Z 200.000,A 0.000,B 0.000,C 180.000,E1 0.000} C_DIS
LIN {X -202.316,Y 64.586,Z 200.000,A 0.000,B 0.000,C 180.000,E1 0.000} C_DIS
LIN {X -205.373,Y 54.086,Z 200.000,A 0.000,B 0.000,C 180.000,E1 0.000} C_DIS
LIN {X -207.885,Y 43.441,Z 200.000,A 0.000,B 0.000,C 180.000,E1 0.000} C_DIS
LIN {X -209.847,Y 32.683,Z 200.000,A 0.000,B 0.000,C 180.000,E1 0.000} C_DIS
LIN {X -211.250,Y 21.836,Z 200.000,A 0.000,B 0.000,C 180.000,E1 0.000} C_DIS
LIN {X -212.095,Y 10.933,Z 200.000,A 0.000,B 0.000,C 180.000,E1 0.000} C_DIS
LIN {X -212.375,Y 0.000,Z 200.000,A 0.000,B 0.000,C 180.000,E1 0.000} C_DIS
LIN {X -212.095,Y -10.933,Z 200.000,A 0.000,B 0.000,C 180.000,E1 0.000} C_DIS
LIN {X -211.250,Y -21.836,Z 200.000,A 0.000,B 0.000,C 180.000,E1 0.000} C_DIS
LIN {X -209.847,Y -32.683,Z 200.000,A 0.000,B 0.000,C 180.000,E1 0.000} C_DIS
LIN {X -207.885,Y -43.441,Z 200.000,A 0.000,B 0.000,C 180.000,E1 0.000} C_DIS
LIN {X -205.373,Y -54.086,Z 200.000,A 0.000,B 0.000,C 180.000,E1 0.000} C_DIS
LIN {X -202.316,Y -64.586,Z 200.000,A 0.000,B 0.000,C 180.000,E1 0.000} C_DIS
LIN {X -198.724,Y -74.916,Z 200.000,A 0.000,B 0.000,C 180.000,E1 0.000} C_DIS
LIN {X -194.604,Y -85.046,Z 200.000,A 0.000,B 0.000,C 180.000,E1 0.000} C_DIS
LIN {X -189.967,Y -94.951,Z 200.000,A 0.000,B 0.000,C 180.000,E1 0.000} C_DIS
LIN {X -184.828,Y -104.605,Z 200.000,A 0.000,B 0.000,C 180.000,E1 0.000} C_DIS
LIN {X -179.197,Y -113.982,Z 200.000,A 0.000,B 0.000,C 180.000,E1 0.000} C_DIS
LIN {X -173.092,Y -123.055,Z 200.000,A 0.000,B 0.000,C 180.000,E1 0.000} C_DIS
LIN {X -166.527,Y -131.803,Z 200.000,A 0.000,B 0.000,C 180.000,E1 0.000} C_DIS
LIN {X -159.522,Y -140.201,Z 200.000,A 0.000,B 0.000,C 180.000,E1 0.000} C_DIS
LIN {X -152.094,Y -148.226,Z 200.000,A 0.000,B 0.000,C 180.000,E1 0.000} C_DIS
LIN {X -144.261,Y -155.859,Z 200.000,A 0.000,B 0.000,C 180.000,E1 0.000} C_DIS
LIN {X -136.047,Y -163.079,Z 200.000,A 0.000,B 0.000,C 180.000,E1 0.000} C_DIS
LIN {X -127.471,Y -169.866,Z 200.000,A 0.000,B 0.000,C 180.000,E1 0.000} C_DIS
LIN {X -118.557,Y -176.204,Z 200.000,A 0.000,B 0.000,C 180.000,E1 0.000} C_DIS
LIN {X -109.329,Y -182.073,Z 200.000,A 0.000,B 0.000,C 180.000,E1 0.000} C_DIS
LIN {X -99.811,Y -187.460,Z 200.000,A 0.000,B 0.000,C 180.000,E1 0.000} C_DIS
LIN {X -90.029,Y -192.349,Z 200.000,A 0.000,B 0.000,C 180.000,E1 0.000} C_DIS
LIN {X -80.008,Y -196.730,Z 200.000,A 0.000,B 0.000,C 180.000,E1 0.000} C_DIS
LIN {X -76.010,Y -198.237,Z 200.000,A 0.000,B 0.000,C 180.000,E1 0.000} C_DIS
LIN {X -69.774,Y -200.587,Z 200.000,A 0.000,B 0.000,C 180.000,E1 0.000} C_DIS
LIN {X -59.356,Y -203.913,Z 200.000,A 0.000,B 0.000,C 180.000,E1 0.000} C_DIS
LIN {X -48.780,Y -206.698,Z 200.000,A 0.000,B 0.000,C 180.000,E1 0.000} C_DIS
LIN {X -38.075,Y -208.934,Z 200.000,A 0.000,B 0.000,C 180.000,E1 0.000} C_DIS
LIN {X -27.269,Y -210.617,Z 200.000,A 0.000,B 0.000,C 180.000,E1 0.000} C_DIS
LIN {X -16.389,Y -211.742,Z 200.000,A 0.000,B 0.000,C 180.000,E1 0.000} C_DIS
LIN {X -5.468,Y -212.306,Z 200.000,A 0.000,B 0.000,C 180.000,E1 0.000} C_DIS
LIN {X 5.468,Y -212.306,Z 200.000,A 0.000,B 0.000,C 180.000,E1 0.000} C_DIS
LIN {X 16.389,Y -211.742,Z 200.000,A 0.000,B 0.000,C 180.000,E1 0.000} C_DIS
LIN {X 27.269,Y -210.617,Z 200.000,A 0.000,B 0.000,C 180.000,E1 0.000} C_DIS
LIN {X 38.075,Y -208.934,Z 200.000,A 0.000,B 0.000,C 180.000,E1 0.000} C_DIS
;rapid-leaky
$VEL.CP=0.3
LIN {X 35.288,Y -193.641,Z 200.000,A 0.000,B 0.000,C 180.000,E1 0.000} C_DIS
;bead-perimeter_inner
$VEL.CP=0.49
LIN {X 45.210,Y -191.568,Z 200.000,A 0.000,B 0.000,C 180.000,E1 0.000} C_DIS
LIN {X 55.012,Y -188.987,Z 200.000,A 0.000,B 0.000,C 180.000,E1 0.000} C_DIS
LIN {X 64.667,Y -185.904,Z 200.000,A 0.000,B 0.000,C 180.000,E1 0.000} C_DIS
LIN {X 74.152,Y -182.329,Z 200.000,A 0.000,B 0.000,C 180.000,E1 0.000} C_DIS
LIN {X 83.439,Y -178.270,Z 200.000,A 0.000,B 0.000,C 180.000,E1 0.000} C_DIS
LIN {X 92.505,Y -173.739,Z 200.000,A 0.000,B 0.000,C 180.000,E1 0.000} C_DIS
LIN {X 101.326,Y -168.746,Z 200.000,A 0.000,B 0.000,C 180.000,E1 0.000} C_DIS
LIN {X 109.879,Y -163.306,Z 200.000,A 0.000,B 0.000,C 180.000,E1 0.000} C_DIS
LIN {X 118.141,Y -157.432,Z 200.000,A 0.000,B 0.000,C 180.000,E1 0.000} C_DIS
LIN {X 126.090,Y -151.142,Z 200.000,A 0.000,B 0.000,C 180.000,E1 0.000} C_DIS
LIN {X 133.702,Y -144.451,Z 200.000,A 0.000,B 0.000,C 180.000,E1 0.000} C_DIS
LIN {X 140.961,Y -137.377,Z 200.000,A 0.000,B 0.000,C 180.000,E1 0.000} C_DIS
LIN {X 147.845,Y -129.939,Z 200.000,A 0.000,B 0.000,C 180.000,E1 0.000} C_DIS
LIN {X 154.338,Y -122.155,Z 200.000,A 0.000,B 0.000,C 180.000,E1 0.000} C_DIS
LIN {X 160.422,Y -114.048,Z 200.000,A 0.000,B 0.000,C 180.000,E1 0.000} C_DIS
LIN {X 166.080,Y -105.639,Z 200.000,A 0.000,B 0.000,C 180.000,E1 0.000} C_DIS
LIN {X 171.299,Y -96.949,Z 200.000,A 0.000,B 0.000,C 180.000,E1 0.000} C_DIS
LIN {X 176.062,Y -88.002,Z 200.000,A 0.000,B 0.000,C 180.000,E1 0.000} C_DIS
LIN {X 180.360,Y -78.820,Z 200.000,A 0.000,B 0.000,C 180.000,E1 0.000} C_DIS
LIN {X 184.178,Y -69.433,Z 200.000,A 0.000,B 0.000,C 180.000,E1 0.000} C_DIS
LIN {X 187.507,Y -59.859,Z 200.000,A 0.000,B 0.000,C 180.000,E1 0.000} C_DIS
LIN {X 190.341,Y -50.127,Z 200.000,A 0.000,B 0.000,C 180.000,E1 0.000} C_DIS
LIN {X 192.669,Y -40.261,Z 200.000,A 0.000,B 0.000,C 180.000,E1 0.000} C_DIS
LIN {X 194.487,Y -30.291,Z 200.000,A 0.000,B 0.000,C 180.000,E1 0.000} C_DIS
LIN {X 195.787,Y -20.238,Z 200.000,A 0.000,B 0.000,C 180.000,E1 0.000} C_DIS
LIN {X 196.570,Y -10.133,Z 200.000,A 0.000,B 0.000,C 180.000,E1 0.000} C_DIS
LIN {X 196.830,Y 0.000,Z 200.000,A 0.000,B 0.000,C 180.000,E1 0.000} C_DIS
LIN {X 196.570,Y 10.133,Z 200.000,A 0.000,B 0.000,C 180.000,E1 0.000} C_DIS
LIN {X 195.787,Y 20.238,Z 200.000,A 0.000,B 0.000,C 180.000,E1 0.000} C_DIS
LIN {X 194.487,Y 30.291,Z 200.000,A 0.000,B 0.000,C 180.000,E1 0.000} C_DIS
LIN {X 192.669,Y 40.261,Z 200.000,A 0.000,B 0.000,C 180.000,E1 0.000} C_DIS
LIN {X 190.341,Y 50.127,Z 200.000,A 0.000,B 0.000,C 180.000,E1 0.000} C_DIS
LIN {X 187.507,Y 59.859,Z 200.000,A 0.000,B 0.000,C 180.000,E1 0.000} C_DIS
LIN {X 184.178,Y 69.433,Z 200.000,A 0.000,B 0.000,C 180.000,E1 0.000} C_DIS
LIN {X 180.359,Y 78.821,Z 200.000,A 0.000,B 0.000,C 180.000,E1 0.000} C_DIS
LIN {X 178.718,Y 82.327,Z 200.000,A 0.000,B 0.000,C 180.000,E1 0.000} C_DIS
LIN {X 176.062,Y 88.001,Z 200.000,A 0.000,B 0.000,C 180.000,E1 0.000} C_DIS
LIN {X 171.299,Y 96.949,Z 200.000,A 0.000,B 0.000,C 180.000,E1 0.000} C_DIS
LIN {X 166.080,Y 105.639,Z 200.000,A 0.000,B 0.000,C 180.000,E1 0.000} C_DIS
LIN {X 160.422,Y 114.048,Z 200.000,A 0.000,B 0.000,C 180.000,E1 0.000} C_DIS
LIN {X 154.338,Y 122.155,Z 200.000,A 0.000,B 0.000,C 180.000,E1 0.000} C_DIS
LIN {X 147.845,Y 129.939,Z 200.000,A 0.000,B 0.000,C 180.000,E1 0.000} C_DIS
LIN {X 140.961,Y 137.377,Z 200.000,A 0.000,B 0.000,C 180.000,E1 0.000} C_DIS
LIN {X 133.702,Y 144.451,Z 200.000,A 0.000,B 0.000,C 180.000,E1 0.000} C_DIS
LIN {X 126.090,Y 151.142,Z 200.000,A 0.000,B 0.000,C 180.000,E1 0.000} C_DIS
LIN {X 118.141,Y 157.432,Z 200.000,A 0.000,B 0.000,C 180.000,E1 0.000} C_DIS
LIN {X 109.879,Y 163.306,Z 200.000,A 0.000,B 0.000,C 180.000,E1 0.000} C_DIS
LIN {X 101.326,Y 168.746,Z 200.000,A 0.000,B 0.000,C 180.000,E1 0.000} C_DIS
LIN {X 92.505,Y 173.739,Z 200.000,A 0.000,B 0.000,C 180.000,E1 0.000} C_DIS
LIN {X 83.439,Y 178.270,Z 200.000,A 0.000,B 0.000,C 180.000,E1 0.000} C_DIS
LIN {X 74.151,Y 182.330,Z 200.000,A 0.000,B 0.000,C 180.000,E1 0.000} C_DIS
LIN {X 70.530,Y 183.695,Z 200.000,A 0.000,B 0.000,C 180.000,E1 0.000} C_DIS
LIN {X 64.668,Y 185.904,Z 200.000,A 0.000,B 0.000,C 180.000,E1 0.000} C_DIS
LIN {X 55.012,Y 188.987,Z 200.000,A 0.000,B 0.000,C 180.000,E1 0.000} C_DIS
LIN {X 45.210,Y 191.568,Z 200.000,A 0.000,B 0.000,C 180.000,E1 0.000} C_DIS
LIN {X 35.288,Y 193.641,Z 200.000,A 0.000,B 0.000,C 180.000,E1 0.000} C_DIS
LIN {X 25.272,Y 195.201,Z 200.000,A 0.000,B 0.000,C 180.000,E1 0.000} C_DIS
LIN {X 15.189,Y 196.244,Z 200.000,A 0.000,B 0.000,C 180.000,E1 0.000} C_DIS
LIN {X 5.067,Y 196.766,Z 200.000,A 0.000,B 0.000,C 180.000,E1 0.000} C_DIS
LIN {X -5.067,Y 196.766,Z 200.000,A 0.000,B 0.000,C 180.000,E1 0.000} C_DIS
LIN {X -15.189,Y 196.244,Z 200.000,A 0.000,B 0.000,C 180.000,E1 0.000} C_DIS
LIN {X -25.272,Y 195.201,Z 200.000,A 0.000,B 0.000,C 180.000,E1 0.000} C_DIS
LIN {X -35.288,Y 193.641,Z 200.000,A 0.000,B 0.000,C 180.000,E1 0.000} C_DIS
LIN {X -45.210,Y 191.568,Z 200.000,A 0.000,B 0.000,C 180.000,E1 0.000} C_DIS
LIN {X -55.012,Y 188.987,Z 200.000,A 0.000,B 0.000,C 180.000,E1 0.000} C_DIS
LIN {X -64.667,Y 185.904,Z 200.000,A 0.000,B 0.000,C 180.000,E1 0.000} C_DIS
LIN {X -74.152,Y 182.329,Z 200.000,A 0.000,B 0.000,C 180.000,E1 0.000} C_DIS
LIN {X -83.439,Y 178.270,Z 200.000,A 0.000,B 0.000,C 180.000,E1 0.000} C_DIS
LIN {X -92.505,Y 173.739,Z 200.000,A 0.000,B 0.000,C 180.000,E1 0.000} C_DIS
LIN {X -101.326,Y 168.746,Z 200.000,A 0.000,B 0.000,C 180.000,E1 0.000} C_DIS
LIN {X -109.879,Y 163.306,Z 200.000,A 0.000,B 0.000,C 180.000,E1 0.000} C_DIS
LIN {X -118.141,Y 157.432,Z 200.000,A 0.000,B 0.000,C 180.000,E1 0.000} C_DIS
LIN {X -126.090,Y 151.142,Z 200.000,A 0.000,B 0.000,C 180.000,E1 0.000} C_DIS
LIN {X -133.702,Y 144.451,Z 200.000,A 0.000,B 0.000,C 180.000,E1 0.000} C_DIS
LIN {X -140.961,Y 137.377,Z 200.000,A 0.000,B 0.000,C 180.000,E1 0.000} C_DIS
LIN {X -147.845,Y 129.939,Z 200.000,A 0.000,B 0.000,C 180.000,E1 0.000} C_DIS
LIN {X -154.338,Y 122.155,Z 200.000,A 0.000,B 0.000,C 180.000,E1 0.000} C_DIS
LIN {X -160.422,Y 114.048,Z 200.000,A 0.000,B 0.000,C 180.000,E1 0.000} C_DIS
LIN {X -166.080,Y 105.639,Z 200.000,A 0.000,B 0.000,C 180.000,E1 0.000} C_DIS
LIN {X -171.299,Y 96.949,Z 200.000,A 0.000,B 0.000,C 180.000,E1 0.000} C_DIS
LIN {X -176.062,Y 88.002,Z 200.000,A 0.000,B 0.000,C 180.000,E1 0.000} C_DIS
LIN {X -180.360,Y 78.820,Z 200.000,A 0.000,B 0.000,C 180.000,E1 0.000} C_DIS
LIN {X -184.178,Y 69.433,Z 200.000,A 0.000,B 0.000,C 180.000,E1 0.000} C_DIS
LIN {X -187.507,Y 59.859,Z 200.000,A 0.000,B 0.000,C 180.000,E1 0.000} C_DIS
LIN {X -190.341,Y 50.127,Z 200.000,A 0.000,B 0.000,C 180.000,E1 0.000} C_DIS
LIN {X -192.669,Y 40.261,Z 200.000,A 0.000,B 0.000,C 180.000,E1 0.000} C_DIS
LIN {X -194.487,Y 30.291,Z 200.000,A 0.000,B 0.000,C 180.000,E1 0.000} C_DIS
LIN {X -195.787,Y 20.238,Z 200.000,A 0.000,B 0.000,C 180.000,E1 0.000} C_DIS
LIN {X -196.570,Y 10.133,Z 200.000,A 0.000,B 0.000,C 180.000,E1 0.000} C_DIS
LIN {X -196.830,Y 0.000,Z 200.000,A 0.000,B 0.000,C 180.000,E1 0.000} C_DIS
LIN {X -196.570,Y -10.133,Z 200.000,A 0.000,B 0.000,C 180.000,E1 0.000} C_DIS
LIN {X -195.787,Y -20.238,Z 200.000,A 0.000,B 0.000,C 180.000,E1 0.000} C_DIS
LIN {X -194.487,Y -30.291,Z 200.000,A 0.000,B 0.000,C 180.000,E1 0.000} C_DIS
LIN {X -192.669,Y -40.261,Z 200.000,A 0.000,B 0.000,C 180.000,E1 0.000} C_DIS
LIN {X -190.341,Y -50.127,Z 200.000,A 0.000,B 0.000,C 180.000,E1 0.000} C_DIS
LIN {X -187.507,Y -59.859,Z 200.000,A 0.000,B 0.000,C 180.000,E1 0.000} C_DIS
LIN {X -184.178,Y -69.433,Z 200.000,A 0.000,B 0.000,C 180.000,E1 0.000} C_DIS
LIN {X -180.359,Y -78.821,Z 200.000,A 0.000,B 0.000,C 180.000,E1 0.000} C_DIS
LIN {X -176.062,Y -88.001,Z 200.000,A 0.000,B 0.000,C 180.000,E1 0.000} C_DIS
LIN {X -171.299,Y -96.949,Z 200.000,A 0.000,B 0.000,C 180.000,E1 0.000} C_DIS
LIN {X -166.080,Y -105.639,Z 200.000,A 0.000,B 0.000,C 180.000,E1 0.000} C_DIS
LIN {X -160.422,Y -114.048,Z 200.000,A 0.000,B 0.000,C 180.000,E1 0.000} C_DIS
LIN {X -154.338,Y -122.155,Z 200.000,A 0.000,B 0.000,C 180.000,E1 0.000} C_DIS
LIN {X -147.845,Y -129.939,Z 200.000,A 0.000,B 0.000,C 180.000,E1 0.000} C_DIS
LIN {X -140.961,Y -137.377,Z 200.000,A 0.000,B 0.000,C 180.000,E1 0.000} C_DIS
LIN {X -133.702,Y -144.451,Z 200.000,A 0.000,B 0.000,C 180.000,E1 0.000} C_DIS
LIN {X -126.090,Y -151.142,Z 200.000,A 0.000,B 0.000,C 180.000,E1 0.000} C_DIS
LIN {X -118.141,Y -157.432,Z 200.000,A 0.000,B 0.000,C 180.000,E1 0.000} C_DIS
LIN {X -109.879,Y -163.306,Z 200.000,A 0.000,B 0.000,C 180.000,E1 0.000} C_DIS
LIN {X -101.326,Y -168.746,Z 200.000,A 0.000,B 0.000,C 180.000,E1 0.000} C_DIS
LIN {X -92.505,Y -173.739,Z 200.000,A 0.000,B 0.000,C 180.000,E1 0.000} C_DIS
LIN {X -83.439,Y -178.270,Z 200.000,A 0.000,B 0.000,C 180.000,E1 0.000} C_DIS
LIN {X -74.151,Y -182.330,Z 200.000,A 0.000,B 0.000,C 180.000,E1 0.000} C_DIS
LIN {X -70.530,Y -183.695,Z 200.000,A 0.000,B 0.000,C 180.000,E1 0.000} C_DIS
LIN {X -64.668,Y -185.904,Z 200.000,A 0.000,B 0.000,C 180.000,E1 0.000} C_DIS
LIN {X -55.012,Y -188.987,Z 200.000,A 0.000,B 0.000,C 180.000,E1 0.000} C_DIS
LIN {X -45.210,Y -191.568,Z 200.000,A 0.000,B 0.000,C 180.000,E1 0.000} C_DIS
LIN {X -35.288,Y -193.641,Z 200.000,A 0.000,B 0.000,C 180.000,E1 0.000} C_DIS
LIN {X -25.272,Y -195.201,Z 200.000,A 0.000,B 0.000,C 180.000,E1 0.000} C_DIS
LIN {X -15.189,Y -196.244,Z 200.000,A 0.000,B 0.000,C 180.000,E1 0.000} C_DIS
LIN {X -5.067,Y -196.766,Z 200.000,A 0.000,B 0.000,C 180.000,E1 0.000} C_DIS
LIN {X 5.067,Y -196.766,Z 200.000,A 0.000,B 0.000,C 180.000,E1 0.000} C_DIS
LIN {X 15.189,Y -196.244,Z 200.000,A 0.000,B 0.000,C 180.000,E1 0.000} C_DIS
LIN {X 25.272,Y -195.201,Z 200.000,A 0.000,B 0.000,C 180.000,E1 0.000} C_DIS
LIN {X 35.288,Y -193.641,Z 200.000,A 0.000,B 0.000,C 180.000,E1 0.000} C_DIS
;rapid-leaky
$VEL.CP=0.3
LIN {X -47.142,Y -172.694,Z 200.000,A 0.000,B 0.000,C 180.000,E1 0.000} C_DIS
;bead-sparse_infill
$VEL.CP=0.49
LIN {X 172.708,Y 47.157,Z 200.000,A 0.000,B 0.000,C 180.000,E1 0.000} C_DIS
LIN {X 170.583,Y 54.456,Z 200.000,A 0.000,B 0.000,C 180.000,E1 0.000} C_DIS
LIN {X 167.554,Y 63.166,Z 200.000,A 0.000,B 0.000,C 180.000,E1 0.000} C_DIS
LIN {X 164.080,Y 71.706,Z 200.000,A 0.000,B 0.000,C 180.000,E1 0.000} C_DIS
LIN {X 162.634,Y 74.797,Z 200.000,A 0.000,B 0.000,C 180.000,E1 0.000} C_DIS
LIN {X 160.171,Y 80.058,Z 200.000,A 0.000,B 0.000,C 180.000,E1 0.000} C_DIS
LIN {X 155.837,Y 88.198,Z 200.000,A 0.000,B 0.000,C 180.000,E1 0.000} C_DIS
LIN {X 151.090,Y 96.104,Z 200.000,A 0.000,B 0.000,C 180.000,E1 0.000} C_DIS
LIN {X 145.943,Y 103.754,Z 200.000,A 0.000,B 0.000,C 180.000,E1 0.000} C_DIS
LIN {X 140.408,Y 111.129,Z 200.000,A 0.000,B 0.000,C 180.000,E1 0.000} C_DIS
LIN {X 134.500,Y 118.211,Z 200.000,A 0.000,B 0.000,C 180.000,E1 0.000} C_DIS
LIN {X 128.238,Y 124.977,Z 200.000,A 0.000,B 0.000,C 180.000,E1 0.000} C_DIS
LIN {X 121.634,Y 131.413,Z 200.000,A 0.000,B 0.000,C 180.000,E1 0.000} C_DIS
LIN {X 114.709,Y 137.500,Z 200.000,A 0.000,B 0.000,C 180.000,E1 0.000} C_DIS
LIN {X 109.888,Y 141.314,Z 200.000,A 0.000,B 0.000,C 180.000,E1 0.000} C_DIS
LIN {X -141.328,Y -109.903,Z 200.000,A 0.000,B 0.000,C 180.000,E1 0.000} C_DIS
LIN {X -145.943,Y -103.754,Z 200.000,A 0.000,B 0.000,C 180.000,E1 0.000} C_DIS
LIN {X -151.090,Y -96.104,Z 200.000,A 0.000,B 0.000,C 180.000,E1 0.000} C_DIS
LIN {X -155.837,Y -88.198,Z 200.000,A 0.000,B 0.000,C 180.000,E1 0.000} C_DIS
LIN {X -160.171,Y -80.058,Z 200.000,A 0.000,B 0.000,C 180.000,E1 0.000} C_DIS
LIN {X -164.081,Y -71.706,Z 200.000,A 0.000,B 0.000,C 180.000,E1 0.000} C_DIS
LIN {X -167.554,Y -63.166,Z 200.000,A 0.000,B 0.000,C 180.000,E1 0.000} C_DIS
LIN {X -170.583,Y -54.456,Z 200.000,A 0.000,B 0.000,C 180.000,E1 0.000} C_DIS
LIN {X -173.161,Y -45.602,Z 200.000,A 0.000,B 0.000,C 180.000,E1 0.000} C_DIS
LIN {X -175.279,Y -36.627,Z 200.000,A 0.000,B 0.000,C 180.000,E1 0.000} C_DIS
LIN {X -176.932,Y -27.557,Z 200.000,A 0.000,B 0.000,C 180.000,E1 0.000} C_DIS
LIN {X -178.116,Y -18.411,Z 200.000,A 0.000,B 0.000,C 180.000,E1 0.000} C_DIS
LIN {X -178.828,Y -9.218,Z 200.000,A 0.000,B 0.000,C 180.000,E1 0.000} C_DIS
LIN {X -179.064,Y 0.000,Z 200.000,A 0.000,B 0.000,C 180.000,E1 0.000} C_DIS
LIN {X -178.828,Y 9.218,Z 200.000,A 0.000,B 0.000,C 180.000,E1 0.000} C_DIS
LIN {X -178.798,Y 9.605,Z 200.000,A 0.000,B 0.000,C 180.000,E1 0.000} C_DIS
LIN {X -9.658,Y 178.745,Z 200.000,A 0.000,B 0.000,C 180.000,E1 0.000} C_DIS
;rapid-leaky
$VEL.CP=0.3
LIN {X -198.727,Y -41.527,Z 210.000,A 0.000,B 0.000,C 180.000,E1 0.000} C_DIS
;bead-perimeter_outer
$VEL.CP=0.48
LIN {X -196.326,Y -51.703,Z 210.000,A 0.000,B 0.000,C 180.000,E1 0.000} C_DIS
LIN {X -193.403,Y -61.741,Z 210.000,A 0.000,B 0.000,C 180.000,E1 0.000} C_DIS
LIN {X -189.968,Y -71.617,Z 210.000,A 0.000,B 0.000,C 180.000,E1 0.000} C_DIS
LIN {X -186.031,Y -81.300,Z 210.000,A 0.000,B 0.000,C 180.000,E1 0.000} C_DIS
LIN {X -181.598,Y -90.768,Z 210.000,A 0.000,B 0.000,C 180.000,E1 0.000} C_DIS
LIN {X -176.685,Y -99.997,Z 210.000,A 0.000,B 0.000,C 180.000,E1 0.000} C_DIS
LIN {X -171.303,Y -108.960,Z 210.000,A 0.000,B 0.000,C 180.000,E1 0.000} C_DIS
LIN {X -165.466,Y -117.634,Z 210.000,A 0.000,B 0.000,C 180.000,E1 0.000} C_DIS
LIN {X -159.192,Y -125.996,Z 210.000,A 0.000,B 0.000,C 180.000,E1 0.000} C_DIS
LIN {X -152.494,Y -134.024,Z 210.000,A 0.000,B 0.000,C 180.000,E1 0.000} C_DIS
LIN {X -145.393,Y -141.696,Z 210.000,A 0.000,B 0.000,C 180.000,E1 0.000} C_DIS
LIN {X -137.906,Y -148.993,Z 210.000,A 0.000,B 0.000,C 180.000,E1 0.000} C_DIS
LIN {X -130.053,Y -155.895,Z 210.000,A 0.000,B 0.000,C 180.000,E1 0.000} C_DIS
LIN {X -121.854,Y -162.383,Z 210.000,A 0.000,B 0.000,C 180.000,E1 0.000} C_DIS
LIN {X -113.334,Y -168.441,Z 210.000,A 0.000,B 0.000,C 180.000,E1 0.000} C_DIS
LIN {X -104.513,Y -174.052,Z 210.000,A 0.000,B 0.000,C 180.000,E1 0.000} C_DIS
LIN {X -95.414,Y -179.201,Z 210.000,A 0.000,B 0.000,C 180.000,E1 0.000} C_DIS
LIN {X -86.063,Y -183.875,Z 210.000,A 0.000,B 0.000,C 180.000,E1 0.000} C_DIS
LIN {X -76.482,Y -188.062,Z 210.000,A 0.000,B 0.000,C 180.000,E1 0.000} C_DIS
LIN {X -66.701,Y -191.750,Z 210.000,A 0.000,B 0.000,C 180.000,E1 0.000} C_DIS
LIN {X -56.742,Y -194.929,Z 210.000,A 0.000,B 0.000,C 180.000,E1 0.000} C_DIS
LIN {X -46.632,Y -197.591,Z 210.000,A 0.000,B 0.000,C 180.000,E1 0.000} C_DIS
LIN {X -36.397,Y -199.730,Z 210.000,A 0.000,B 0.000,C 180.000,E1 0.000} C_DIS
LIN {X -26.068,Y -201.339,Z 210.000,A 0.000,B 0.000,C 180.000,E1 0.000} C_DIS
LIN {X -15.668,Y -202.413,Z 210.000,A 0.000,B 0.000,C 180.000,E1 0.000} C_DIS
LIN {X -5.228,Y -202.952,Z 210.000,A 0.000,B 0.000,C 180.000,E1 0.000} C_DIS
LIN {X 5.228,Y -202.952,Z 210.000,A 0.000,B 0.000,C 180.000,E1 0.000} C_DIS
LIN {X 15.668,Y -202.413,Z 210.000,A 0.000,B 0.000,C 180.000,E1 0.000} C_DIS
LIN {X 26.068,Y -201.339,Z 210.000,A 0.000,B 0.000,C 180.000,E1 0.000} C_DIS
LIN {X 36.397,Y -199.730,Z 210.000,A 0.000,B 0.000,C 180.000,E1 0.000} C_DIS
LIN {X 46.632,Y -197.591,Z 210.000,A 0.000,B 0.000,C 180.000,E1 0.000} C_DIS
LIN {X 56.742,Y -194.929,Z 210.000,A 0.000,B 0.000,C 180.000,E1 0.000} C_DIS
LIN {X 66.701,Y -191.750,Z 210.000,A 0.000,B 0.000,C 180.000,E1 0.000} C_DIS
LIN {X 76.483,Y -188.061,Z 210.000,A 0.000,B 0.000,C 180.000,E1 0.000} C_DIS
LIN {X 86.063,Y -183.875,Z 210.000,A 0.000,B 0.000,C 180.000,E1 0.000} C_DIS
LIN {X 95.414,Y -179.201,Z 210.000,A 0.000,B 0.000,C 180.000,E1 0.000} C_DIS
LIN {X 104.513,Y -174.052,Z 210.000,A 0.000,B 0.000,C 180.000,E1 0.000} C_DIS
LIN {X 113.334,Y -168.441,Z 210.000,A 0.000,B 0.000,C 180.000,E1 0.000} C_DIS
LIN {X 121.854,Y -162.383,Z 210.000,A 0.000,B 0.000,C 180.000,E1 0.000} C_DIS
LIN {X 130.053,Y -155.895,Z 210.000,A 0.000,B 0.000,C 180.000,E1 0.000} C_DIS
LIN {X 137.906,Y -148.993,Z 210.000,A 0.000,B 0.000,C 180.000,E1 0.000} C_DIS
LIN {X 145.393,Y -141.696,Z 210.000,A 0.000,B 0.000,C 180.000,E1 0.000} C_DIS
LIN {X 152.493,Y -134.024,Z 210.000,A 0.000,B 0.000,C 180.000,E1 0.000} C_DIS
LIN {X 159.192,Y -125.996,Z 210.000,A 0.000,B 0.000,C 180.000,E1 0.000} C_DIS
LIN {X 165.466,Y -117.634,Z 210.000,A 0.000,B 0.000,C 180.000,E1 0.000} C_DIS
LIN {X 171.303,Y -108.960,Z 210.000,A 0.000,B 0.000,C 180.000,E1 0.000} C_DIS
LIN {X 176.685,Y -99.997,Z 210.000,A 0.000,B 0.000,C 180.000,E1 0.000} C_DIS
LIN {X 181.598,Y -90.768,Z 210.000,A 0.000,B 0.000,C 180.000,E1 0.000} C_DIS
LIN {X 186.031,Y -81.300,Z 210.000,A 0.000,B 0.000,C 180.000,E1 0.000} C_DIS
LIN {X 189.968,Y -71.617,Z 210.000,A 0.000,B 0.000,C 180.000,E1 0.000} C_DIS
LIN {X 193.403,Y -61.741,Z 210.000,A 0.000,B 0.000,C 180.000,E1 0.000} C_DIS
LIN {X 196.326,Y -51.703,Z 210.000,A 0.000,B 0.000,C 180.000,E1 0.000} C_DIS
LIN {X 198.727,Y -41.527,Z 210.000,A 0.000,B 0.000,C 180.000,E1 0.000} C_DIS
LIN {X 200.602,Y -31.244,Z 210.000,A 0.000,B 0.000,C 180.000,E1 0.000} C_DIS
LIN {X 201.943,Y -20.874,Z 210.000,A 0.000,B 0.000,C 180.000,E1 0.000} C_DIS
LIN {X 202.751,Y -10.450,Z 210.000,A 0.000,B 0.000,C 180.000,E1 0.000} C_DIS
LIN {X 203.019,Y 0.000,Z 210.000,A 0.000,B 0.000,C 180.000,E1 0.000} C_DIS
LIN {X 202.751,Y 10.450,Z 210.000,A 0.000,B 0.000,C 180.000,E1 0.000} C_DIS
LIN {X 201.943,Y 20.874,Z 210.000,A 0.000,B 0.000,C 180.000,E1 0.000} C_DIS
LIN {X 200.602,Y 31.244,Z 210.000,A 0.000,B 0.000,C 180.000,E1 0.000} C_DIS
LIN {X 198.727,Y 41.527,Z 210.000,A 0.000,B 0.000,C 180.000,E1 0.000} C_DIS
LIN {X 196.326,Y 51.703,Z 210.000,A 0.000,B 0.000,C 180.000,E1 0.000} C_DIS
LIN {X 193.403,Y 61.741,Z 210.000,A 0.000,B 0.000,C 180.000,E1 0.000} C_DIS
LIN {X 189.968,Y 71.617,Z 210.000,A 0.000,B 0.000,C 180.000,E1 0.000} C_DIS
LIN {X 186.031,Y 81.300,Z 210.000,A 0.000,B 0.000,C 180.000,E1 0.000} C_DIS
LIN {X 181.598,Y 90.768,Z 210.000,A 0.000,B 0.000,C 180.000,E1 0.000} C_DIS
LIN {X 176.685,Y 99.997,Z 210.000,A 0.000,B 0.000,C 180.000,E1 0.000} C_DIS
LIN {X 171.303,Y 108.960,Z 210.000,A 0.000,B 0.000,C 180.000,E1 0.000} C_DIS
LIN {X 165.466,Y 117.634,Z 210.000,A 0.000,B 0.000,C 180.000,E1 0.000} C_DIS
LIN {X 159.192,Y 125.996,Z 210.000,A 0.000,B 0.000,C 180.000,E1 0.000} C_DIS
LIN {X 152.494,Y 134.024,Z 210.000,A 0.000,B 0.000,C 180.000,E1 0.000} C_DIS
LIN {X 145.393,Y 141.696,Z 210.000,A 0.000,B 0.000,C 180.000,E1 0.000} C_DIS
LIN {X 137.906,Y 148.993,Z 210.000,A 0.000,B 0.000,C 180.000,E1 0.000} C_DIS
LIN {X 130.053,Y 155.895,Z 210.000,A 0.000,B 0.000,C 180.000,E1 0.000} C_DIS
LIN {X 121.854,Y 162.383,Z 210.000,A 0.000,B 0.000,C 180.000,E1 0.000} C_DIS
LIN {X 113.334,Y 168.441,Z 210.000,A 0.000,B 0.000,C 180.000,E1 0.000} C_DIS
LIN {X 104.513,Y 174.052,Z 210.000,A 0.000,B 0.000,C 180.000,E1 0.000} C_DIS
LIN {X 95.414,Y 179.201,Z 210.000,A 0.000,B 0.000,C 180.000,E1 0.000} C_DIS
LIN {X 86.063,Y 183.875,Z 210.000,A 0.000,B 0.000,C 180.000,E1 0.000} C_DIS
LIN {X 76.482,Y 188.062,Z 210.000,A 0.000,B 0.000,C 180.000,E1 0.000} C_DIS
LIN {X 66.701,Y 191.750,Z 210.000,A 0.000,B 0.000,C 180.000,E1 0.000} C_DIS
LIN {X 56.742,Y 194.929,Z 210.000,A 0.000,B 0.000,C 180.000,E1 0.000} C_DIS
LIN {X 46.632,Y 197.591,Z 210.000,A 0.000,B 0.000,C 180.000,E1 0.000} C_DIS
LIN {X 36.397,Y 199.730,Z 210.000,A 0.000,B 0.000,C 180.000,E1 0.000} C_DIS
LIN {X 26.068,Y 201.339,Z 210.000,A 0.000,B 0.000,C 180.000,E1 0.000} C_DIS
LIN {X 15.668,Y 202.413,Z 210.000,A 0.000,B 0.000,C 180.000,E1 0.000} C_DIS
LIN {X 5.228,Y 202.952,Z 210.000,A 0.000,B 0.000,C 180.000,E1 0.000} C_DIS
LIN {X -5.228,Y 202.952,Z 210.000,A 0.000,B 0.000,C 180.000,E1 0.000} C_DIS
LIN {X -15.668,Y 202.413,Z 210.000,A 0.000,B 0.000,C 180.000,E1 0.000} C_DIS
LIN {X -26.068,Y 201.339,Z 210.000,A 0.000,B 0.000,C 180.000,E1 0.000} C_DIS
LIN {X -36.397,Y 199.730,Z 210.000,A 0.000,B 0.000,C 180.000,E1 0.000} C_DIS
LIN {X -46.632,Y 197.591,Z 210.000,A 0.000,B 0.000,C 180.000,E1 0.000} C_DIS
LIN {X -56.742,Y 194.929,Z 210.000,A 0.000,B 0.000,C 180.000,E1 0.000} C_DIS
LIN {X -66.701,Y 191.750,Z 210.000,A 0.000,B 0.000,C 180.000,E1 0.000} C_DIS
LIN {X -76.483,Y 188.061,Z 210.000,A 0.000,B 0.000,C 180.000,E1 0.000} C_DIS
LIN {X -86.063,Y 183.875,Z 210.000,A 0.000,B 0.000,C 180.000,E1 0.000} C_DIS
LIN {X -95.414,Y 179.201,Z 210.000,A 0.000,B 0.000,C 180.000,E1 0.000} C_DIS
LIN {X -104.513,Y 174.052,Z 210.000,A 0.000,B 0.000,C 180.000,E1 0.000} C_DIS
LIN {X -113.334,Y 168.441,Z 210.000,A 0.000,B 0.000,C 180.000,E1 0.000} C_DIS
LIN {X -121.854,Y 162.383,Z 210.000,A 0.000,B 0.000,C 180.000,E1 0.000} C_DIS
LIN {X -130.053,Y 155.895,Z 210.000,A 0.000,B 0.000,C 180.000,E1 0.000} C_DIS
LIN {X -137.906,Y 148.993,Z 210.000,A 0.000,B 0.000,C 180.000,E1 0.000} C_DIS
LIN {X -145.393,Y 141.696,Z 210.000,A 0.000,B 0.000,C 180.000,E1 0.000} C_DIS
LIN {X -152.493,Y 134.024,Z 210.000,A 0.000,B 0.000,C 180.000,E1 0.000} C_DIS
LIN {X -159.192,Y 125.996,Z 210.000,A 0.000,B 0.000,C 180.000,E1 0.000} C_DIS
LIN {X -165.466,Y 117.634,Z 210.000,A 0.000,B 0.000,C 180.000,E1 0.000} C_DIS
LIN {X -171.303,Y 108.960,Z 210.000,A 0.000,B 0.000,C 180.000,E1 0.000} C_DIS
LIN {X -176.685,Y 99.997,Z 210.000,A 0.000,B 0.000,C 180.000,E1 0.000} C_DIS
LIN {X -181.598,Y 90.768,Z 210.000,A 0.000,B 0.000,C 180.000,E1 0.000} C_DIS
LIN {X -186.031,Y 81.300,Z 210.000,A 0.000,B 0.000,C 180.000,E1 0.000} C_DIS
LIN {X -189.968,Y 71.617,Z 210.000,A 0.000,B 0.000,C 180.000,E1 0.000} C_DIS
LIN {X -193.403,Y 61.741,Z 210.000,A 0.000,B 0.000,C 180.000,E1 0.000} C_DIS
LIN {X -196.326,Y 51.703,Z 210.000,A 0.000,B 0.000,C 180.000,E1 0.000} C_DIS
LIN {X -198.727,Y 41.527,Z 210.000,A 0.000,B 0.000,C 180.000,E1 0.000} C_DIS
LIN {X -200.602,Y 31.244,Z 210.000,A 0.000,B 0.000,C 180.000,E1 0.000} C_DIS
LIN {X -201.943,Y 20.874,Z 210.000,A 0.000,B 0.000,C 180.000,E1 0.000} C_DIS
LIN {X -202.751,Y 10.450,Z 210.000,A 0.000,B 0.000,C 180.000,E1 0.000} C_DIS
LIN {X -203.019,Y 0.000,Z 210.000,A 0.000,B 0.000,C 180.000,E1 0.000} C_DIS
LIN {X -202.751,Y -10.450,Z 210.000,A 0.000,B 0.000,C 180.000,E1 0.000} C_DIS
LIN {X -201.943,Y -20.874,Z 210.000,A 0.000,B 0.000,C 180.000,E1 0.000} C_DIS
LIN {X -200.602,Y -31.244,Z 210.000,A 0.000,B 0.000,C 180.000,E1 0.000} C_DIS
LIN {X -198.727,Y -41.527,Z 210.000,A 0.000,B 0.000,C 180.000,E1 0.000} C_DIS
;rapid-leaky
$VEL.CP=0.3
LIN {X -183.511,Y -38.347,Z 210.000,A 0.000,B 0.000,C 180.000,E1 0.000} C_DIS
;bead-perimeter_inner
$VEL.CP=0.48
LIN {X -181.293,Y -47.744,Z 210.000,A 0.000,B 0.000,C 180.000,E1 0.000} C_DIS
LIN {X -178.595,Y -57.013,Z 210.000,A 0.000,B 0.000,C 180.000,E1 0.000} C_DIS
LIN {X -175.422,Y -66.133,Z 210.000,A 0.000,B 0.000,C 180.000,E1 0.000} C_DIS
LIN {X -171.786,Y -75.075,Z 210.000,A 0.000,B 0.000,C 180.000,E1 0.000} C_DIS
